KUKA KRL data list: CNC2.dat

&ACCESS RV
DEFDAT CNC2 Public
DECL GLOBAL FRAME gfCNCPoint2[30000]


gfCNCPoint2[1] = {X 204.1061, Y 40.0576, Z -2.1667, A 0.000, B 0.000, C 0.000 }
gfCNCPoint2[2] = {X 204.4089, Y 40.9162, Z -2.1667, A 0.000, B 0.000, C 0.000 }
gfCNCPoint2[3] = {X 204.5137, Y 41.8206, Z -2.1667, A 0.000, B 0.000, C 0.000 }
gfCNCPoint2[4] = {X 204.4154, Y 42.7257, Z -2.1667, A 0.000, B 0.000, C 0.000 }
gfCNCPoint2[5] = {X 204.1188, Y 43.5864, Z -2.1667, A 0.000, B 0.000, C 0.000 }
gfCNCPoint2[6] = {X 203.6387, Y 44.3600, Z -2.1667, A 0.000, B 0.000, C 0.000 }
gfCNCPoint2[7] = {X 202.9990, Y 45.0078, Z -2.1667, A 0.000, B 0.000, C 0.000 }
gfCNCPoint2[8] = {X 202.4628, Y 45.4414, Z -2.1667, A 0.000, B 0.000, C 0.000 }
gfCNCPoint2[9] = {X 201.7788, Y 45.8885, Z -2.1667, A 0.000, B 0.000, C 0.000 }
gfCNCPoint2[10] = {X 201.0196, Y 46.1910, Z -2.1667, A 0.000, B 0.000, C 0.000 }
gfCNCPoint2[11] = {X 200.2155, Y 46.3368, Z -2.1667, A 0.000, B 0.000, C 0.000 }
gfCNCPoint2[12] = {X 199.3985, Y 46.3200, Z -2.1667, A 0.000, B 0.000, C 0.000 }
gfCNCPoint2[13] = {X 198.6011, Y 46.1413, Z -2.1667, A 0.000, B 0.000, C 0.000 }
gfCNCPoint2[14] = {X 196.8579, Y 47.0738, Z -2.1667, A 0.000, B 0.000, C 0.000 }
gfCNCPoint2[15] = {X 195.0540, Y 47.8828, Z -2.1667, A 0.000, B 0.000, C 0.000 }
gfCNCPoint2[16] = {X 193.1983, Y 48.5643, Z -2.1667, A 0.000, B 0.000, C 0.000 }
gfCNCPoint2[17] = {X 191.2996, Y 49.1151, Z -2.1667, A 0.000, B 0.000, C 0.000 }
gfCNCPoint2[18] = {X 189.3771, Y 49.5045, Z -2.1667, A 0.000, B 0.000, C 0.000 }
gfCNCPoint2[19] = {X 187.4280, Y 49.7244, Z -2.1667, A 0.000, B 0.000, C 0.000 }
gfCNCPoint2[20] = {X 185.4671, Y 49.7730, Z -2.1667, A 0.000, B 0.000, C 0.000 }
gfCNCPoint2[21] = {X 183.5094, Y 49.6499, Z -2.1667, A 0.000, B 0.000, C 0.000 }
gfCNCPoint2[22] = {X 181.5700, Y 49.3561, Z -2.1667, A 0.000, B 0.000, C 0.000 }
gfCNCPoint2[23] = {X 179.7098, Y 48.8912, Z -2.1667, A 0.000, B 0.000, C 0.000 }
gfCNCPoint2[24] = {X 177.9148, Y 48.2172, Z -2.1667, A 0.000, B 0.000, C 0.000 }
gfCNCPoint2[25] = {X 176.2082, Y 47.3431, Z -2.1667, A 0.000, B 0.000, C 0.000 }
gfCNCPoint2[26] = {X 174.6124, Y 46.2802, Z -2.1667, A 0.000, B 0.000, C 0.000 }
gfCNCPoint2[27] = {X 173.4016, Y 45.2583, Z -2.1667, A 0.000, B 0.000, C 0.000 }
gfCNCPoint2[28] = {X 172.3241, Y 44.0965, Z -2.1667, A 0.000, B 0.000, C 0.000 }
gfCNCPoint2[29] = {X 171.3961, Y 42.8123, Z -2.1667, A 0.000, B 0.000, C 0.000 }
gfCNCPoint2[30] = {X 170.6313, Y 41.4246, Z -2.1667, A 0.000, B 0.000, C 0.000 }
gfCNCPoint2[31] = {X 170.0410, Y 39.9542, Z -2.1667, A 0.000, B 0.000, C 0.000 }
gfCNCPoint2[32] = {X 169.6341, Y 38.4229, Z -2.1667, A 0.000, B 0.000, C 0.000 }
gfCNCPoint2[33] = {X 169.4166, Y 36.8534, Z -2.1667, A 0.000, B 0.000, C 0.000 }
gfCNCPoint2[34] = {X 169.3333, Y 35.0485, Z -2.1667, A 0.000, B 0.000, C 0.000 }
gfCNCPoint2[35] = {X 169.4768, Y 33.2475, Z -2.1667, A 0.000, B 0.000, C 0.000 }
gfCNCPoint2[36] = {X 169.8448, Y 31.4786, Z -2.1667, A 0.000, B 0.000, C 0.000 }
gfCNCPoint2[37] = {X 170.4315, Y 29.7697, Z -2.1667, A 0.000, B 0.000, C 0.000 }
gfCNCPoint2[38] = {X 171.1150, Y 28.3909, Z -2.1667, A 0.000, B 0.000, C 0.000 }
gfCNCPoint2[39] = {X 171.9904, Y 27.1252, Z -2.1667, A 0.000, B 0.000, C 0.000 }
gfCNCPoint2[40] = {X 173.0396, Y 25.9993, Z -2.1667, A 0.000, B 0.000, C 0.000 }
gfCNCPoint2[41] = {X 174.2404, Y 25.0368, Z -2.1667, A 0.000, B 0.000, C 0.000 }
gfCNCPoint2[42] = {X 175.5677, Y 24.2579, Z -2.1667, A 0.000, B 0.000, C 0.000 }
gfCNCPoint2[43] = {X 174.6553, Y 23.9382, Z -2.1667, A 0.000, B 0.000, C 0.000 }
gfCNCPoint2[44] = {X 173.8439, Y 23.4129, Z -2.1667, A 0.000, B 0.000, C 0.000 }
gfCNCPoint2[45] = {X 173.1787, Y 22.7114, Z -2.1667, A 0.000, B 0.000, C 0.000 }
gfCNCPoint2[46] = {X 172.6973, Y 21.8731, Z -2.1667, A 0.000, B 0.000, C 0.000 }
gfCNCPoint2[47] = {X 171.3803, Y 18.6480, Z -2.1667, A 0.000, B 0.000, C 0.000 }
gfCNCPoint2[48] = {X 167.6770, Y 20.1603, Z -2.1667, A 0.000, B 0.000, C 0.000 }
gfCNCPoint2[49] = {X 167.6769, Y 20.1601, Z -2.1667, A 0.000, B 0.000, C 0.000 }
gfCNCPoint2[50] = {X 171.4542, Y 18.6179, Z -2.1667, A 0.000, B 0.000, C 0.000 }
gfCNCPoint2[51] = {X 170.1367, Y 15.3911, Z -2.1667, A 0.000, B 0.000, C 0.000 }
gfCNCPoint2[52] = {X 169.8835, Y 14.4675, Z -2.1667, A 0.000, B 0.000, C 0.000 }
gfCNCPoint2[53] = {X 169.8570, Y 13.5102, Z -2.1667, A 0.000, B 0.000, C 0.000 }
gfCNCPoint2[54] = {X 170.0588, Y 12.5740, Z -2.1667, A 0.000, B 0.000, C 0.000 }
gfCNCPoint2[55] = {X 170.4774, Y 11.7127, Z -2.1667, A 0.000, B 0.000, C 0.000 }
gfCNCPoint2[56] = {X 171.0888, Y 10.9755, Z -2.1667, A 0.000, B 0.000, C 0.000 }
gfCNCPoint2[57] = {X 171.8578, Y 10.4048, Z -2.1667, A 0.000, B 0.000, C 0.000 }
gfCNCPoint2[58] = {X 172.4867, Y 10.0462, Z -2.1667, A 0.000, B 0.000, C 0.000 }
gfCNCPoint2[59] = {X 173.3363, Y 9.6929, Z -2.1667, A 0.000, B 0.000, C 0.000 }
gfCNCPoint2[60] = {X 174.2443, Y 9.5431, Z -2.1667, A 0.000, B 0.000, C 0.000 }
gfCNCPoint2[61] = {X 175.1624, Y 9.6048, Z -2.1667, A 0.000, B 0.000, C 0.000 }
gfCNCPoint2[62] = {X 176.0421, Y 9.8746, Z -2.1667, A 0.000, B 0.000, C 0.000 }
gfCNCPoint2[63] = {X 178.2221, Y 8.9431, Z -2.1667, A 0.000, B 0.000, C 0.000 }
gfCNCPoint2[64] = {X 180.4850, Y 8.2365, Z -2.1667, A 0.000, B 0.000, C 0.000 }
gfCNCPoint2[65] = {X 182.8078, Y 7.7622, Z -2.1667, A 0.000, B 0.000, C 0.000 }
gfCNCPoint2[66] = {X 185.1665, Y 7.5249, Z -2.1667, A 0.000, B 0.000, C 0.000 }
gfCNCPoint2[67] = {X 187.5372, Y 7.5270, Z -2.1667, A 0.000, B 0.000, C 0.000 }
gfCNCPoint2[68] = {X 189.8955, Y 7.7686, Z -2.1667, A 0.000, B 0.000, C 0.000 }
gfCNCPoint2[69] = {X 191.6205, Y 8.1236, Z -2.1667, A 0.000, B 0.000, C 0.000 }
gfCNCPoint2[70] = {X 193.3000, Y 8.6537, Z -2.1667, A 0.000, B 0.000, C 0.000 }
gfCNCPoint2[71] = {X 194.9162, Y 9.3534, Z -2.1667, A 0.000, B 0.000, C 0.000 }
gfCNCPoint2[72] = {X 196.4521, Y 10.2153, Z -2.1667, A 0.000, B 0.000, C 0.000 }
gfCNCPoint2[73] = {X 197.8914, Y 11.2302, Z -2.1667, A 0.000, B 0.000, C 0.000 }
gfCNCPoint2[74] = {X 199.1662, Y 12.3971, Z -2.1667, A 0.000, B 0.000, C 0.000 }
gfCNCPoint2[75] = {X 200.2713, Y 13.7259, Z -2.1667, A 0.000, B 0.000, C 0.000 }
gfCNCPoint2[76] = {X 201.1862, Y 15.1921, Z -2.1667, A 0.000, B 0.000, C 0.000 }
gfCNCPoint2[77] = {X 201.8941, Y 16.7687, Z -2.1667, A 0.000, B 0.000, C 0.000 }
gfCNCPoint2[78] = {X 202.3577, Y 18.3894, Z -2.1667, A 0.000, B 0.000, C 0.000 }
gfCNCPoint2[79] = {X 202.6328, Y 20.0525, Z -2.1667, A 0.000, B 0.000, C 0.000 }
gfCNCPoint2[80] = {X 202.7157, Y 21.7361, Z -2.1667, A 0.000, B 0.000, C 0.000 }
gfCNCPoint2[81] = {X 202.6054, Y 23.4182, Z -2.1667, A 0.000, B 0.000, C 0.000 }
gfCNCPoint2[82] = {X 202.3032, Y 25.0766, Z -2.1667, A 0.000, B 0.000, C 0.000 }
gfCNCPoint2[83] = {X 201.8258, Y 26.6078, Z -2.1667, A 0.000, B 0.000, C 0.000 }
gfCNCPoint2[84] = {X 201.1376, Y 28.0565, Z -2.1667, A 0.000, B 0.000, C 0.000 }
gfCNCPoint2[85] = {X 200.2525, Y 29.3941, Z -2.1667, A 0.000, B 0.000, C 0.000 }
gfCNCPoint2[86] = {X 199.1879, Y 30.5938, Z -2.1667, A 0.000, B 0.000, C 0.000 }
gfCNCPoint2[87] = {X 197.9652, Y 31.6318, Z -2.1667, A 0.000, B 0.000, C 0.000 }
gfCNCPoint2[88] = {X 198.7272, Y 31.8156, Z -2.1667, A 0.000, B 0.000, C 0.000 }
gfCNCPoint2[89] = {X 199.4387, Y 32.1445, Z -2.1667, A 0.000, B 0.000, C 0.000 }
gfCNCPoint2[90] = {X 200.0724, Y 32.6059, Z -2.1667, A 0.000, B 0.000, C 0.000 }
gfCNCPoint2[91] = {X 200.6039, Y 33.1820, Z -2.1667, A 0.000, B 0.000, C 0.000 }
gfCNCPoint2[92] = {X 201.0129, Y 33.8507, Z -2.1667, A 0.000, B 0.000, C 0.000 }
gfCNCPoint2[93] = {X 204.0341, Y 40.0925, Z -2.1667, A 0.000, B 0.000, C 0.000 }
gfCNCPoint2[94] = {X 204.3309, Y 40.9342, Z -2.1667, A 0.000, B 0.000, C 0.000 }
gfCNCPoint2[95] = {X 204.4337, Y 41.8209, Z -2.1667, A 0.000, B 0.000, C 0.000 }
gfCNCPoint2[96] = {X 204.3373, Y 42.7082, Z -2.1667, A 0.000, B 0.000, C 0.000 }
gfCNCPoint2[97] = {X 204.0465, Y 43.5521, Z -2.1667, A 0.000, B 0.000, C 0.000 }
gfCNCPoint2[98] = {X 203.5758, Y 44.3105, Z -2.1667, A 0.000, B 0.000, C 0.000 }
gfCNCPoint2[99] = {X 202.9487, Y 44.9456, Z -2.1667, A 0.000, B 0.000, C 0.000 }
gfCNCPoint2[100] = {X 202.4125, Y 45.3791, Z -2.1667, A 0.000, B 0.000, C 0.000 }
gfCNCPoint2[101] = {X 201.7355, Y 45.8209, Z -2.1667, A 0.000, B 0.000, C 0.000 }
gfCNCPoint2[102] = {X 200.9837, Y 46.1181, Z -2.1667, A 0.000, B 0.000, C 0.000 }
gfCNCPoint2[103] = {X 200.1877, Y 46.2587, Z -2.1667, A 0.000, B 0.000, C 0.000 }
gfCNCPoint2[104] = {X 199.3796, Y 46.2370, Z -2.1667, A 0.000, B 0.000, C 0.000 }
gfCNCPoint2[105] = {X 198.5922, Y 46.0539, Z -2.1667, A 0.000, B 0.000, C 0.000 }
gfCNCPoint2[106] = {X 196.8470, Y 46.9900, Z -2.1667, A 0.000, B 0.000, C 0.000 }
gfCNCPoint2[107] = {X 195.0406, Y 47.8019, Z -2.1667, A 0.000, B 0.000, C 0.000 }
gfCNCPoint2[108] = {X 193.1819, Y 48.4855, Z -2.1667, A 0.000, B 0.000, C 0.000 }
gfCNCPoint2[109] = {X 191.2800, Y 49.0375, Z -2.1667, A 0.000, B 0.000, C 0.000 }
gfCNCPoint2[110] = {X 189.3644, Y 49.4255, Z -2.1667, A 0.000, B 0.000, C 0.000 }
gfCNCPoint2[111] = {X 187.4222, Y 49.6446, Z -2.1667, A 0.000, B 0.000, C 0.000 }
gfCNCPoint2[112] = {X 185.4683, Y 49.6930, Z -2.1667, A 0.000, B 0.000, C 0.000 }
gfCNCPoint2[113] = {X 183.5177, Y 49.5703, Z -2.1667, A 0.000, B 0.000, C 0.000 }
gfCNCPoint2[114] = {X 181.5852, Y 49.2775, Z -2.1667, A 0.000, B 0.000, C 0.000 }
gfCNCPoint2[115] = {X 179.7338, Y 48.8148, Z -2.1667, A 0.000, B 0.000, C 0.000 }
gfCNCPoint2[116] = {X 177.9472, Y 48.1441, Z -2.1667, A 0.000, B 0.000, C 0.000 }
gfCNCPoint2[117] = {X 176.2487, Y 47.2741, Z -2.1667, A 0.000, B 0.000, C 0.000 }
gfCNCPoint2[118] = {X 174.6604, Y 46.2162, Z -2.1667, A 0.000, B 0.000, C 0.000 }
gfCNCPoint2[119] = {X 173.4568, Y 45.2004, Z -2.1667, A 0.000, B 0.000, C 0.000 }
gfCNCPoint2[120] = {X 172.3859, Y 44.0456, Z -2.1667, A 0.000, B 0.000, C 0.000 }
gfCNCPoint2[121] = {X 171.4634, Y 42.7691, Z -2.1667, A 0.000, B 0.000, C 0.000 }
gfCNCPoint2[122] = {X 170.7033, Y 41.3898, Z -2.1667, A 0.000, B 0.000, C 0.000 }
gfCNCPoint2[123] = {X 170.1166, Y 39.9282, Z -2.1667, A 0.000, B 0.000, C 0.000 }
gfCNCPoint2[124] = {X 169.7123, Y 38.4060, Z -2.1667, A 0.000, B 0.000, C 0.000 }
gfCNCPoint2[125] = {X 169.4962, Y 36.8460, Z -2.1667, A 0.000, B 0.000, C 0.000 }
gfCNCPoint2[126] = {X 169.4132, Y 35.0508, Z -2.1667, A 0.000, B 0.000, C 0.000 }
gfCNCPoint2[127] = {X 169.5559, Y 33.2593, Z -2.1667, A 0.000, B 0.000, C 0.000 }
gfCNCPoint2[128] = {X 169.9219, Y 31.4998, Z -2.1667, A 0.000, B 0.000, C 0.000 }
gfCNCPoint2[129] = {X 170.5055, Y 29.8001, Z -2.1667, A 0.000, B 0.000, C 0.000 }
gfCNCPoint2[130] = {X 171.2085, Y 28.3899, Z -2.1667, A 0.000, B 0.000, C 0.000 }
gfCNCPoint2[131] = {X 172.1139, Y 27.1002, Z -2.1667, A 0.000, B 0.000, C 0.000 }
gfCNCPoint2[132] = {X 173.2013, Y 25.9598, Z -2.1667, A 0.000, B 0.000, C 0.000 }
gfCNCPoint2[133] = {X 174.4465, Y 24.9941, Z -2.1667, A 0.000, B 0.000, C 0.000 }
gfCNCPoint2[134] = {X 175.8218, Y 24.2249, Z -2.1667, A 0.000, B 0.000, C 0.000 }
gfCNCPoint2[135] = {X 175.0307, Y 24.0140, Z -2.1667, A 0.000, B 0.000, C 0.000 }
gfCNCPoint2[136] = {X 174.2991, Y 23.6464, Z -2.1667, A 0.000, B 0.000, C 0.000 }
gfCNCPoint2[137] = {X 173.6577, Y 23.1376, Z -2.1667, A 0.000, B 0.000, C 0.000 }
gfCNCPoint2[138] = {X 173.1333, Y 22.5089, Z -2.1667, A 0.000, B 0.000, C 0.000 }
gfCNCPoint2[139] = {X 172.7479, Y 21.7866, Z -2.1667, A 0.000, B 0.000, C 0.000 }
gfCNCPoint2[140] = {X 171.4542, Y 18.6179, Z -2.1667, A 0.000, B 0.000, C 0.000 }
gfCNCPoint2[141] = {X 167.6769, Y 20.1601, Z -2.1667, A 0.000, B 0.000, C 0.000 }
gfCNCPoint2[142] = {X 167.6769, Y 20.1601, Z 0.8333, A 0.000, B 0.000, C 0.000 }
gfCNCPoint2[143] = {X 167.6769, Y 20.1601, Z 11.0000, A 0.000, B 0.000, C 0.000 }
gfCNCPoint2[144] = {X 210.1659, Y 28.5742, Z 11.0000, A 0.000, B 0.000, C 0.000 }
gfCNCPoint2[145] = {X 210.1659, Y 28.5742, Z 0.8333, A 0.000, B 0.000, C 0.000 }
gfCNCPoint2[146] = {X 210.1659, Y 28.5742, Z -2.1667, A 0.000, B 0.000, C 0.000 }
gfCNCPoint2[147] = {X 214.2459, Y 28.5742, Z -2.1667, A 0.000, B 0.000, C 0.000 }
gfCNCPoint2[148] = {X 214.2459, Y 17.4624, Z -2.1667, A 0.000, B 0.000, C 0.000 }
gfCNCPoint2[149] = {X 214.2405, Y 16.7693, Z -2.1667, A 0.000, B 0.000, C 0.000 }
gfCNCPoint2[150] = {X 214.2433, Y 16.2731, Z -2.1667, A 0.000, B 0.000, C 0.000 }
gfCNCPoint2[151] = {X 213.6052, Y 15.6019, Z -2.1667, A 0.000, B 0.000, C 0.000 }
gfCNCPoint2[152] = {X 213.1248, Y 14.8101, Z -2.1667, A 0.000, B 0.000, C 0.000 }
gfCNCPoint2[153] = {X 212.8241, Y 13.9341, Z -2.1667, A 0.000, B 0.000, C 0.000 }
gfCNCPoint2[154] = {X 212.7172, Y 13.0141, Z -2.1667, A 0.000, B 0.000, C 0.000 }
gfCNCPoint2[155] = {X 212.7170, Y 12.1868, Z -2.1667, A 0.000, B 0.000, C 0.000 }
gfCNCPoint2[156] = {X 212.8253, Y 11.2255, Z -2.1667, A 0.000, B 0.000, C 0.000 }
gfCNCPoint2[157] = {X 213.1448, Y 10.3124, Z -2.1667, A 0.000, B 0.000, C 0.000 }
gfCNCPoint2[158] = {X 213.6595, Y 9.4933, Z -2.1667, A 0.000, B 0.000, C 0.000 }
gfCNCPoint2[159] = {X 214.3435, Y 8.8093, Z -2.1667, A 0.000, B 0.000, C 0.000 }
gfCNCPoint2[160] = {X 215.1626, Y 8.2946, Z -2.1667, A 0.000, B 0.000, C 0.000 }
gfCNCPoint2[161] = {X 216.0757, Y 7.9751, Z -2.1667, A 0.000, B 0.000, C 0.000 }
gfCNCPoint2[162] = {X 217.0370, Y 7.8668, Z -2.1667, A 0.000, B 0.000, C 0.000 }
gfCNCPoint2[163] = {X 223.4805, Y 7.8668, Z -2.1667, A 0.000, B 0.000, C 0.000 }
gfCNCPoint2[164] = {X 224.4418, Y 7.9751, Z -2.1667, A 0.000, B 0.000, C 0.000 }
gfCNCPoint2[165] = {X 225.3549, Y 8.2946, Z -2.1667, A 0.000, B 0.000, C 0.000 }
gfCNCPoint2[166] = {X 226.1740, Y 8.8093, Z -2.1667, A 0.000, B 0.000, C 0.000 }
gfCNCPoint2[167] = {X 226.8580, Y 9.4933, Z -2.1667, A 0.000, B 0.000, C 0.000 }
gfCNCPoint2[168] = {X 227.3727, Y 10.3124, Z -2.1667, A 0.000, B 0.000, C 0.000 }
gfCNCPoint2[169] = {X 227.6922, Y 11.2255, Z -2.1667, A 0.000, B 0.000, C 0.000 }
gfCNCPoint2[170] = {X 227.8005, Y 12.1868, Z -2.1667, A 0.000, B 0.000, C 0.000 }
gfCNCPoint2[171] = {X 227.8005, Y 12.9781, Z -2.1667, A 0.000, B 0.000, C 0.000 }
gfCNCPoint2[172] = {X 227.6991, Y 13.9083, Z -2.1667, A 0.000, B 0.000, C 0.000 }
gfCNCPoint2[173] = {X 227.3998, Y 14.7949, Z -2.1667, A 0.000, B 0.000, C 0.000 }
gfCNCPoint2[174] = {X 226.9167, Y 15.5962, Z -2.1667, A 0.000, B 0.000, C 0.000 }
gfCNCPoint2[175] = {X 226.2723, Y 16.2747, Z -2.1667, A 0.000, B 0.000, C 0.000 }
gfCNCPoint2[176] = {X 226.2732, Y 40.9153, Z -2.1667, A 0.000, B 0.000, C 0.000 }
gfCNCPoint2[177] = {X 226.9108, Y 41.5854, Z -2.1667, A 0.000, B 0.000, C 0.000 }
gfCNCPoint2[178] = {X 227.3912, Y 42.3758, Z -2.1667, A 0.000, B 0.000, C 0.000 }
gfCNCPoint2[179] = {X 227.6923, Y 43.2503, Z -2.1667, A 0.000, B 0.000, C 0.000 }
gfCNCPoint2[180] = {X 227.8003, Y 44.1689, Z -2.1667, A 0.000, B 0.000, C 0.000 }
gfCNCPoint2[181] = {X 227.8005, Y 45.0000, Z -2.1667, A 0.000, B 0.000, C 0.000 }
gfCNCPoint2[182] = {X 227.6922, Y 45.9613, Z -2.1667, A 0.000, B 0.000, C 0.000 }
gfCNCPoint2[183] = {X 227.3727, Y 46.8744, Z -2.1667, A 0.000, B 0.000, C 0.000 }
gfCNCPoint2[184] = {X 226.8580, Y 47.6935, Z -2.1667, A 0.000, B 0.000, C 0.000 }
gfCNCPoint2[185] = {X 226.1740, Y 48.3775, Z -2.1667, A 0.000, B 0.000, C 0.000 }
gfCNCPoint2[186] = {X 225.3549, Y 48.8922, Z -2.1667, A 0.000, B 0.000, C 0.000 }
gfCNCPoint2[187] = {X 224.4418, Y 49.2117, Z -2.1667, A 0.000, B 0.000, C 0.000 }
gfCNCPoint2[188] = {X 223.4805, Y 49.3200, Z -2.1667, A 0.000, B 0.000, C 0.000 }
gfCNCPoint2[189] = {X 217.0370, Y 49.3200, Z -2.1667, A 0.000, B 0.000, C 0.000 }
gfCNCPoint2[190] = {X 216.0805, Y 49.2128, Z -2.1667, A 0.000, B 0.000, C 0.000 }
gfCNCPoint2[191] = {X 215.1715, Y 48.8964, Z -2.1667, A 0.000, B 0.000, C 0.000 }
gfCNCPoint2[192] = {X 214.3551, Y 48.3867, Z -2.1667, A 0.000, B 0.000, C 0.000 }
gfCNCPoint2[193] = {X 213.6718, Y 47.7088, Z -2.1667, A 0.000, B 0.000, C 0.000 }
gfCNCPoint2[194] = {X 213.1556, Y 46.8965, Z -2.1667, A 0.000, B 0.000, C 0.000 }
gfCNCPoint2[195] = {X 212.8320, Y 45.9901, Z -2.1667, A 0.000, B 0.000, C 0.000 }
gfCNCPoint2[196] = {X 212.7172, Y 45.0345, Z -2.1667, A 0.000, B 0.000, C 0.000 }
gfCNCPoint2[197] = {X 212.7170, Y 44.1994, Z -2.1667, A 0.000, B 0.000, C 0.000 }
gfCNCPoint2[198] = {X 212.7890, Y 43.4200, Z -2.1667, A 0.000, B 0.000, C 0.000 }
gfCNCPoint2[199] = {X 213.0024, Y 42.6670, Z -2.1667, A 0.000, B 0.000, C 0.000 }
gfCNCPoint2[200] = {X 213.3500, Y 41.9658, Z -2.1667, A 0.000, B 0.000, C 0.000 }
gfCNCPoint2[201] = {X 213.8202, Y 41.3400, Z -2.1667, A 0.000, B 0.000, C 0.000 }
gfCNCPoint2[202] = {X 214.2415, Y 40.8754, Z -2.1667, A 0.000, B 0.000, C 0.000 }
gfCNCPoint2[203] = {X 214.2459, Y 40.3062, Z -2.1667, A 0.000, B 0.000, C 0.000 }
gfCNCPoint2[204] = {X 214.2459, Y 28.5742, Z -2.1667, A 0.000, B 0.000, C 0.000 }
gfCNCPoint2[205] = {X 210.2459, Y 28.5742, Z -2.1667, A 0.000, B 0.000, C 0.000 }
gfCNCPoint2[206] = {X 214.3259, Y 28.5742, Z -2.1667, A 0.000, B 0.000, C 0.000 }
gfCNCPoint2[207] = {X 214.3259, Y 17.4621, Z -2.1667, A 0.000, B 0.000, C 0.000 }
gfCNCPoint2[208] = {X 214.3205, Y 16.7693, Z -2.1667, A 0.000, B 0.000, C 0.000 }
gfCNCPoint2[209] = {X 214.3235, Y 16.2360, Z -2.1667, A 0.000, B 0.000, C 0.000 }
gfCNCPoint2[210] = {X 213.6857, Y 15.5754, Z -2.1667, A 0.000, B 0.000, C 0.000 }
gfCNCPoint2[211] = {X 213.2051, Y 14.7930, Z -2.1667, A 0.000, B 0.000, C 0.000 }
gfCNCPoint2[212] = {X 212.9042, Y 13.9255, Z -2.1667, A 0.000, B 0.000, C 0.000 }
gfCNCPoint2[213] = {X 212.7972, Y 13.0135, Z -2.1667, A 0.000, B 0.000, C 0.000 }
gfCNCPoint2[214] = {X 212.7970, Y 12.1868, Z -2.1667, A 0.000, B 0.000, C 0.000 }
gfCNCPoint2[215] = {X 212.9033, Y 11.2433, Z -2.1667, A 0.000, B 0.000, C 0.000 }
gfCNCPoint2[216] = {X 213.2169, Y 10.3472, Z -2.1667, A 0.000, B 0.000, C 0.000 }
gfCNCPoint2[217] = {X 213.7220, Y 9.5432, Z -2.1667, A 0.000, B 0.000, C 0.000 }
gfCNCPoint2[218] = {X 214.3934, Y 8.8719, Z -2.1667, A 0.000, B 0.000, C 0.000 }
gfCNCPoint2[219] = {X 215.1973, Y 8.3667, Z -2.1667, A 0.000, B 0.000, C 0.000 }
gfCNCPoint2[220] = {X 216.0935, Y 8.0531, Z -2.1667, A 0.000, B 0.000, C 0.000 }
gfCNCPoint2[221] = {X 217.0370, Y 7.9468, Z -2.1667, A 0.000, B 0.000, C 0.000 }
gfCNCPoint2[222] = {X 223.4805, Y 7.9468, Z -2.1667, A 0.000, B 0.000, C 0.000 }
gfCNCPoint2[223] = {X 224.4240, Y 8.0531, Z -2.1667, A 0.000, B 0.000, C 0.000 }
gfCNCPoint2[224] = {X 225.3201, Y 8.3667, Z -2.1667, A 0.000, B 0.000, C 0.000 }
gfCNCPoint2[225] = {X 226.1241, Y 8.8718, Z -2.1667, A 0.000, B 0.000, C 0.000 }
gfCNCPoint2[226] = {X 226.7954, Y 9.5432, Z -2.1667, A 0.000, B 0.000, C 0.000 }
gfCNCPoint2[227] = {X 227.3006, Y 10.3471, Z -2.1667, A 0.000, B 0.000, C 0.000 }
gfCNCPoint2[228] = {X 227.6142, Y 11.2433, Z -2.1667, A 0.000, B 0.000, C 0.000 }
gfCNCPoint2[229] = {X 227.7205, Y 12.1868, Z -2.1667, A 0.000, B 0.000, C 0.000 }
gfCNCPoint2[230] = {X 227.7205, Y 12.9781, Z -2.1667, A 0.000, B 0.000, C 0.000 }
gfCNCPoint2[231] = {X 227.6190, Y 13.9001, Z -2.1667, A 0.000, B 0.000, C 0.000 }
gfCNCPoint2[232] = {X 227.3195, Y 14.7780, Z -2.1667, A 0.000, B 0.000, C 0.000 }
gfCNCPoint2[233] = {X 226.8362, Y 15.5697, Z -2.1667, A 0.000, B 0.000, C 0.000 }
gfCNCPoint2[234] = {X 226.1923, Y 16.2374, Z -2.1667, A 0.000, B 0.000, C 0.000 }
gfCNCPoint2[235] = {X 226.1932, Y 40.9526, Z -2.1667, A 0.000, B 0.000, C 0.000 }
gfCNCPoint2[236] = {X 226.8304, Y 41.6121, Z -2.1667, A 0.000, B 0.000, C 0.000 }
gfCNCPoint2[237] = {X 227.3109, Y 42.3931, Z -2.1667, A 0.000, B 0.000, C 0.000 }
gfCNCPoint2[238] = {X 227.6122, Y 43.2591, Z -2.1667, A 0.000, B 0.000, C 0.000 }
gfCNCPoint2[239] = {X 227.7203, Y 44.1697, Z -2.1667, A 0.000, B 0.000, C 0.000 }
gfCNCPoint2[240] = {X 227.7205, Y 45.0000, Z -2.1667, A 0.000, B 0.000, C 0.000 }
gfCNCPoint2[241] = {X 227.6142, Y 45.9435, Z -2.1667, A 0.000, B 0.000, C 0.000 }
gfCNCPoint2[242] = {X 227.3006, Y 46.8397, Z -2.1667, A 0.000, B 0.000, C 0.000 }
gfCNCPoint2[243] = {X 226.7954, Y 47.6436, Z -2.1667, A 0.000, B 0.000, C 0.000 }
gfCNCPoint2[244] = {X 226.1241, Y 48.3150, Z -2.1667, A 0.000, B 0.000, C 0.000 }
gfCNCPoint2[245] = {X 225.3201, Y 48.8201, Z -2.1667, A 0.000, B 0.000, C 0.000 }
gfCNCPoint2[246] = {X 224.4240, Y 49.1337, Z -2.1667, A 0.000, B 0.000, C 0.000 }
gfCNCPoint2[247] = {X 223.4805, Y 49.2400, Z -2.1667, A 0.000, B 0.000, C 0.000 }
gfCNCPoint2[248] = {X 217.0370, Y 49.2400, Z -2.1667, A 0.000, B 0.000, C 0.000 }
gfCNCPoint2[249] = {X 216.0982, Y 49.1348, Z -2.1667, A 0.000, B 0.000, C 0.000 }
gfCNCPoint2[250] = {X 215.2061, Y 48.8243, Z -2.1667, A 0.000, B 0.000, C 0.000 }
gfCNCPoint2[251] = {X 214.4048, Y 48.3240, Z -2.1667, A 0.000, B 0.000, C 0.000 }
gfCNCPoint2[252] = {X 213.7341, Y 47.6587, Z -2.1667, A 0.000, B 0.000, C 0.000 }
gfCNCPoint2[253] = {X 213.2275, Y 46.8614, Z -2.1667, A 0.000, B 0.000, C 0.000 }
gfCNCPoint2[254] = {X 212.9099, Y 45.9717, Z -2.1667, A 0.000, B 0.000, C 0.000 }
gfCNCPoint2[255] = {X 212.7972, Y 45.0338, Z -2.1667, A 0.000, B 0.000, C 0.000 }
gfCNCPoint2[256] = {X 212.7970, Y 44.1994, Z -2.1667, A 0.000, B 0.000, C 0.000 }
gfCNCPoint2[257] = {X 212.8676, Y 43.4347, Z -2.1667, A 0.000, B 0.000, C 0.000 }
gfCNCPoint2[258] = {X 213.0770, Y 42.6958, Z -2.1667, A 0.000, B 0.000, C 0.000 }
gfCNCPoint2[259] = {X 213.4181, Y 42.0077, Z -2.1667, A 0.000, B 0.000, C 0.000 }
gfCNCPoint2[260] = {X 213.8795, Y 41.3938, Z -2.1667, A 0.000, B 0.000, C 0.000 }
gfCNCPoint2[261] = {X 214.3213, Y 40.9065, Z -2.1667, A 0.000, B 0.000, C 0.000 }
gfCNCPoint2[262] = {X 214.3259, Y 40.3065, Z -2.1667, A 0.000, B 0.000, C 0.000 }
gfCNCPoint2[263] = {X 214.3259, Y 28.5742, Z -2.1667, A 0.000, B 0.000, C 0.000 }
gfCNCPoint2[264] = {X 210.3259, Y 28.5742, Z -2.1667, A 0.000, B 0.000, C 0.000 }
gfCNCPoint2[265] = {X 214.4059, Y 28.5742, Z -2.1667, A 0.000, B 0.000, C 0.000 }
gfCNCPoint2[266] = {X 214.4059, Y 17.4618, Z -2.1667, A 0.000, B 0.000, C 0.000 }
gfCNCPoint2[267] = {X 214.4005, Y 16.7692, Z -2.1667, A 0.000, B 0.000, C 0.000 }
gfCNCPoint2[268] = {X 214.4038, Y 16.1985, Z -2.1667, A 0.000, B 0.000, C 0.000 }
gfCNCPoint2[269] = {X 213.7663, Y 15.5487, Z -2.1667, A 0.000, B 0.000, C 0.000 }
gfCNCPoint2[270] = {X 213.2855, Y 14.7758, Z -2.1667, A 0.000, B 0.000, C 0.000 }
gfCNCPoint2[271] = {X 212.9843, Y 13.9168, Z -2.1667, A 0.000, B 0.000, C 0.000 }
gfCNCPoint2[272] = {X 212.8772, Y 13.0128, Z -2.1667, A 0.000, B 0.000, C 0.000 }
gfCNCPoint2[273] = {X 212.8770, Y 12.1868, Z -2.1667, A 0.000, B 0.000, C 0.000 }
gfCNCPoint2[274] = {X 212.9813, Y 11.2611, Z -2.1667, A 0.000, B 0.000, C 0.000 }
gfCNCPoint2[275] = {X 213.2890, Y 10.3819, Z -2.1667, A 0.000, B 0.000, C 0.000 }
gfCNCPoint2[276] = {X 213.7846, Y 9.5931, Z -2.1667, A 0.000, B 0.000, C 0.000 }
gfCNCPoint2[277] = {X 214.4433, Y 8.9344, Z -2.1667, A 0.000, B 0.000, C 0.000 }
gfCNCPoint2[278] = {X 215.2321, Y 8.4388, Z -2.1667, A 0.000, B 0.000, C 0.000 }
gfCNCPoint2[279] = {X 216.1113, Y 8.1311, Z -2.1667, A 0.000, B 0.000, C 0.000 }
gfCNCPoint2[280] = {X 217.0370, Y 8.0268, Z -2.1667, A 0.000, B 0.000, C 0.000 }
gfCNCPoint2[281] = {X 223.4805, Y 8.0268, Z -2.1667, A 0.000, B 0.000, C 0.000 }
gfCNCPoint2[282] = {X 224.4062, Y 8.1311, Z -2.1667, A 0.000, B 0.000, C 0.000 }
gfCNCPoint2[283] = {X 225.2854, Y 8.4388, Z -2.1667, A 0.000, B 0.000, C 0.000 }
gfCNCPoint2[284] = {X 226.0742, Y 8.9344, Z -2.1667, A 0.000, B 0.000, C 0.000 }
gfCNCPoint2[285] = {X 226.7329, Y 9.5931, Z -2.1667, A 0.000, B 0.000, C 0.000 }
gfCNCPoint2[286] = {X 227.2285, Y 10.3819, Z -2.1667, A 0.000, B 0.000, C 0.000 }
gfCNCPoint2[287] = {X 227.5362, Y 11.2611, Z -2.1667, A 0.000, B 0.000, C 0.000 }
gfCNCPoint2[288] = {X 227.6405, Y 12.1868, Z -2.1667, A 0.000, B 0.000, C 0.000 }
gfCNCPoint2[289] = {X 227.6405, Y 12.9781, Z -2.1667, A 0.000, B 0.000, C 0.000 }
gfCNCPoint2[290] = {X 227.5389, Y 13.8918, Z -2.1667, A 0.000, B 0.000, C 0.000 }
gfCNCPoint2[291] = {X 227.2391, Y 14.7609, Z -2.1667, A 0.000, B 0.000, C 0.000 }
gfCNCPoint2[292] = {X 226.7557, Y 15.5429, Z -2.1667, A 0.000, B 0.000, C 0.000 }
gfCNCPoint2[293] = {X 226.1123, Y 16.1997, Z -2.1667, A 0.000, B 0.000, C 0.000 }
gfCNCPoint2[294] = {X 226.1132, Y 40.9903, Z -2.1667, A 0.000, B 0.000, C 0.000 }
gfCNCPoint2[295] = {X 226.7499, Y 41.6390, Z -2.1667, A 0.000, B 0.000, C 0.000 }
gfCNCPoint2[296] = {X 227.2306, Y 42.4105, Z -2.1667, A 0.000, B 0.000, C 0.000 }
gfCNCPoint2[297] = {X 227.5321, Y 43.2680, Z -2.1667, A 0.000, B 0.000, C 0.000 }
gfCNCPoint2[298] = {X 227.6403, Y 44.1704, Z -2.1667, A 0.000, B 0.000, C 0.000 }
gfCNCPoint2[299] = {X 227.6405, Y 45.0000, Z -2.1667, A 0.000, B 0.000, C 0.000 }
gfCNCPoint2[300] = {X 227.5362, Y 45.9257, Z -2.1667, A 0.000, B 0.000, C 0.000 }
gfCNCPoint2[301] = {X 227.2285, Y 46.8050, Z -2.1667, A 0.000, B 0.000, C 0.000 }
gfCNCPoint2[302] = {X 226.7329, Y 47.5937, Z -2.1667, A 0.000, B 0.000, C 0.000 }
gfCNCPoint2[303] = {X 226.0742, Y 48.2524, Z -2.1667, A 0.000, B 0.000, C 0.000 }
gfCNCPoint2[304] = {X 225.2854, Y 48.7480, Z -2.1667, A 0.000, B 0.000, C 0.000 }
gfCNCPoint2[305] = {X 224.4062, Y 49.0557, Z -2.1667, A 0.000, B 0.000, C 0.000 }
gfCNCPoint2[306] = {X 223.4805, Y 49.1600, Z -2.1667, A 0.000, B 0.000, C 0.000 }
gfCNCPoint2[307] = {X 217.0370, Y 49.1600, Z -2.1667, A 0.000, B 0.000, C 0.000 }
gfCNCPoint2[308] = {X 216.1160, Y 49.0568, Z -2.1667, A 0.000, B 0.000, C 0.000 }
gfCNCPoint2[309] = {X 215.2406, Y 48.7521, Z -2.1667, A 0.000, B 0.000, C 0.000 }
gfCNCPoint2[310] = {X 214.4544, Y 48.2613, Z -2.1667, A 0.000, B 0.000, C 0.000 }
gfCNCPoint2[311] = {X 213.7965, Y 47.6085, Z -2.1667, A 0.000, B 0.000, C 0.000 }
gfCNCPoint2[312] = {X 213.2993, Y 46.8263, Z -2.1667, A 0.000, B 0.000, C 0.000 }
gfCNCPoint2[313] = {X 212.9877, Y 45.9534, Z -2.1667, A 0.000, B 0.000, C 0.000 }
gfCNCPoint2[314] = {X 212.8771, Y 45.0332, Z -2.1667, A 0.000, B 0.000, C 0.000 }
gfCNCPoint2[315] = {X 212.8770, Y 44.1994, Z -2.1667, A 0.000, B 0.000, C 0.000 }
gfCNCPoint2[316] = {X 212.9463, Y 43.4493, Z -2.1667, A 0.000, B 0.000, C 0.000 }
gfCNCPoint2[317] = {X 213.1517, Y 42.7246, Z -2.1667, A 0.000, B 0.000, C 0.000 }
gfCNCPoint2[318] = {X 213.4863, Y 42.0497, Z -2.1667, A 0.000, B 0.000, C 0.000 }
gfCNCPoint2[319] = {X 213.9387, Y 41.4475, Z -2.1667, A 0.000, B 0.000, C 0.000 }
gfCNCPoint2[320] = {X 214.4010, Y 40.9376, Z -2.1667, A 0.000, B 0.000, C 0.000 }
gfCNCPoint2[321] = {X 214.4059, Y 40.3068, Z -2.1667, A 0.000, B 0.000, C 0.000 }
gfCNCPoint2[322] = {X 214.4059, Y 28.5742, Z -2.1667, A 0.000, B 0.000, C 0.000 }
gfCNCPoint2[323] = {X 210.4059, Y 28.5742, Z -2.1667, A 0.000, B 0.000, C 0.000 }
gfCNCPoint2[324] = {X 214.4859, Y 28.5742, Z -2.1667, A 0.000, B 0.000, C 0.000 }
gfCNCPoint2[325] = {X 214.4859, Y 17.4614, Z -2.1667, A 0.000, B 0.000, C 0.000 }
gfCNCPoint2[326] = {X 214.4805, Y 16.7691, Z -2.1667, A 0.000, B 0.000, C 0.000 }
gfCNCPoint2[327] = {X 214.4840, Y 16.1605, Z -2.1667, A 0.000, B 0.000, C 0.000 }
gfCNCPoint2[328] = {X 214.4262, Y 16.1133, Z -2.1667, A 0.000, B 0.000, C 0.000 }
gfCNCPoint2[329] = {X 214.3692, Y 16.0650, Z -2.1667, A 0.000, B 0.000, C 0.000 }
gfCNCPoint2[330] = {X 213.7783, Y 15.4331, Z -2.1667, A 0.000, B 0.000, C 0.000 }
gfCNCPoint2[331] = {X 213.3340, Y 14.6908, Z -2.1667, A 0.000, B 0.000, C 0.000 }
gfCNCPoint2[332] = {X 213.0561, Y 13.8716, Z -2.1667, A 0.000, B 0.000, C 0.000 }
gfCNCPoint2[333] = {X 212.9572, Y 13.0121, Z -2.1667, A 0.000, B 0.000, C 0.000 }
gfCNCPoint2[334] = {X 212.9570, Y 12.1868, Z -2.1667, A 0.000, B 0.000, C 0.000 }
gfCNCPoint2[335] = {X 213.0593, Y 11.2789, Z -2.1667, A 0.000, B 0.000, C 0.000 }
gfCNCPoint2[336] = {X 213.3611, Y 10.4166, Z -2.1667, A 0.000, B 0.000, C 0.000 }
gfCNCPoint2[337] = {X 213.8471, Y 9.6430, Z -2.1667, A 0.000, B 0.000, C 0.000 }
gfCNCPoint2[338] = {X 214.4932, Y 8.9969, Z -2.1667, A 0.000, B 0.000, C 0.000 }
gfCNCPoint2[339] = {X 215.2668, Y 8.5109, Z -2.1667, A 0.000, B 0.000, C 0.000 }
gfCNCPoint2[340] = {X 216.1291, Y 8.2091, Z -2.1667, A 0.000, B 0.000, C 0.000 }
gfCNCPoint2[341] = {X 217.0370, Y 8.1068, Z -2.1667, A 0.000, B 0.000, C 0.000 }
gfCNCPoint2[342] = {X 223.4805, Y 8.1068, Z -2.1667, A 0.000, B 0.000, C 0.000 }
gfCNCPoint2[343] = {X 224.3884, Y 8.2091, Z -2.1667, A 0.000, B 0.000, C 0.000 }
gfCNCPoint2[344] = {X 225.2507, Y 8.5109, Z -2.1667, A 0.000, B 0.000, C 0.000 }
gfCNCPoint2[345] = {X 226.0243, Y 8.9969, Z -2.1667, A 0.000, B 0.000, C 0.000 }
gfCNCPoint2[346] = {X 226.6704, Y 9.6430, Z -2.1667, A 0.000, B 0.000, C 0.000 }
gfCNCPoint2[347] = {X 227.1564, Y 10.4166, Z -2.1667, A 0.000, B 0.000, C 0.000 }
gfCNCPoint2[348] = {X 227.4582, Y 11.2789, Z -2.1667, A 0.000, B 0.000, C 0.000 }
gfCNCPoint2[349] = {X 227.5605, Y 12.1868, Z -2.1667, A 0.000, B 0.000, C 0.000 }
gfCNCPoint2[350] = {X 227.5605, Y 12.9781, Z -2.1667, A 0.000, B 0.000, C 0.000 }
gfCNCPoint2[351] = {X 227.4587, Y 13.8835, Z -2.1667, A 0.000, B 0.000, C 0.000 }
gfCNCPoint2[352] = {X 227.1586, Y 14.7437, Z -2.1667, A 0.000, B 0.000, C 0.000 }
gfCNCPoint2[353] = {X 226.6751, Y 15.5159, Z -2.1667, A 0.000, B 0.000, C 0.000 }
gfCNCPoint2[354] = {X 226.0323, Y 16.1615, Z -2.1667, A 0.000, B 0.000, C 0.000 }
gfCNCPoint2[355] = {X 226.0332, Y 41.0286, Z -2.1667, A 0.000, B 0.000, C 0.000 }
gfCNCPoint2[356] = {X 226.1409, Y 41.1154, Z -2.1667, A 0.000, B 0.000, C 0.000 }
gfCNCPoint2[357] = {X 226.7342, Y 41.7472, Z -2.1667, A 0.000, B 0.000, C 0.000 }
gfCNCPoint2[358] = {X 227.1807, Y 42.4899, Z -2.1667, A 0.000, B 0.000, C 0.000 }
gfCNCPoint2[359] = {X 227.4603, Y 43.3103, Z -2.1667, A 0.000, B 0.000, C 0.000 }
gfCNCPoint2[360] = {X 227.5603, Y 44.1712, Z -2.1667, A 0.000, B 0.000, C 0.000 }
gfCNCPoint2[361] = {X 227.5605, Y 45.0000, Z -2.1667, A 0.000, B 0.000, C 0.000 }
gfCNCPoint2[362] = {X 227.4582, Y 45.9079, Z -2.1667, A 0.000, B 0.000, C 0.000 }
gfCNCPoint2[363] = {X 227.1564, Y 46.7702, Z -2.1667, A 0.000, B 0.000, C 0.000 }
gfCNCPoint2[364] = {X 226.6704, Y 47.5438, Z -2.1667, A 0.000, B 0.000, C 0.000 }
gfCNCPoint2[365] = {X 226.0243, Y 48.1899, Z -2.1667, A 0.000, B 0.000, C 0.000 }
gfCNCPoint2[366] = {X 225.2507, Y 48.6760, Z -2.1667, A 0.000, B 0.000, C 0.000 }
gfCNCPoint2[367] = {X 224.3884, Y 48.9777, Z -2.1667, A 0.000, B 0.000, C 0.000 }
gfCNCPoint2[368] = {X 223.4805, Y 49.0800, Z -2.1667, A 0.000, B 0.000, C 0.000 }
gfCNCPoint2[369] = {X 217.0370, Y 49.0800, Z -2.1667, A 0.000, B 0.000, C 0.000 }
gfCNCPoint2[370] = {X 216.1337, Y 48.9787, Z -2.1667, A 0.000, B 0.000, C 0.000 }
gfCNCPoint2[371] = {X 215.2752, Y 48.6800, Z -2.1667, A 0.000, B 0.000, C 0.000 }
gfCNCPoint2[372] = {X 214.5041, Y 48.1986, Z -2.1667, A 0.000, B 0.000, C 0.000 }
gfCNCPoint2[373] = {X 213.8588, Y 47.5584, Z -2.1667, A 0.000, B 0.000, C 0.000 }
gfCNCPoint2[374] = {X 213.3712, Y 46.7912, Z -2.1667, A 0.000, B 0.000, C 0.000 }
gfCNCPoint2[375] = {X 213.0656, Y 45.9351, Z -2.1667, A 0.000, B 0.000, C 0.000 }
gfCNCPoint2[376] = {X 212.9571, Y 45.0325, Z -2.1667, A 0.000, B 0.000, C 0.000 }
gfCNCPoint2[377] = {X 212.9570, Y 44.1994, Z -2.1667, A 0.000, B 0.000, C 0.000 }
gfCNCPoint2[378] = {X 213.0249, Y 43.4640, Z -2.1667, A 0.000, B 0.000, C 0.000 }
gfCNCPoint2[379] = {X 213.2263, Y 42.7534, Z -2.1667, A 0.000, B 0.000, C 0.000 }
gfCNCPoint2[380] = {X 213.5544, Y 42.0917, Z -2.1667, A 0.000, B 0.000, C 0.000 }
gfCNCPoint2[381] = {X 213.9980, Y 41.5012, Z -2.1667, A 0.000, B 0.000, C 0.000 }
gfCNCPoint2[382] = {X 214.4808, Y 40.9687, Z -2.1667, A 0.000, B 0.000, C 0.000 }
gfCNCPoint2[383] = {X 214.4859, Y 40.3072, Z -2.1667, A 0.000, B 0.000, C 0.000 }
gfCNCPoint2[384] = {X 214.4859, Y 28.5742, Z -2.1667, A 0.000, B 0.000, C 0.000 }
gfCNCPoint2[385] = {X 210.4859, Y 28.5742, Z -2.1667, A 0.000, B 0.000, C 0.000 }
gfCNCPoint2[386] = {X 214.5659, Y 28.5742, Z -2.1667, A 0.000, B 0.000, C 0.000 }
gfCNCPoint2[387] = {X 214.5659, Y 17.4611, Z -2.1667, A 0.000, B 0.000, C 0.000 }
gfCNCPoint2[388] = {X 214.5605, Y 16.7687, Z -2.1667, A 0.000, B 0.000, C 0.000 }
gfCNCPoint2[389] = {X 214.5598, Y 16.1862, Z -2.1667, A 0.000, B 0.000, C 0.000 }
gfCNCPoint2[390] = {X 214.5756, Y 16.1310, Z -2.1667, A 0.000, B 0.000, C 0.000 }
gfCNCPoint2[391] = {X 214.4978, Y 16.0687, Z -2.1667, A 0.000, B 0.000, C 0.000 }
gfCNCPoint2[392] = {X 214.4215, Y 16.0044, Z -2.1667, A 0.000, B 0.000, C 0.000 }
gfCNCPoint2[393] = {X 213.8372, Y 15.3783, Z -2.1667, A 0.000, B 0.000, C 0.000 }
gfCNCPoint2[394] = {X 213.3996, Y 14.6420, Z -2.1667, A 0.000, B 0.000, C 0.000 }
gfCNCPoint2[395] = {X 213.1287, Y 13.8295, Z -2.1667, A 0.000, B 0.000, C 0.000 }
gfCNCPoint2[396] = {X 213.0370, Y 12.9779, Z -2.1667, A 0.000, B 0.000, C 0.000 }
gfCNCPoint2[397] = {X 213.0370, Y 12.1868, Z -2.1667, A 0.000, B 0.000, C 0.000 }
gfCNCPoint2[398] = {X 213.1373, Y 11.2967, Z -2.1667, A 0.000, B 0.000, C 0.000 }
gfCNCPoint2[399] = {X 213.4331, Y 10.4513, Z -2.1667, A 0.000, B 0.000, C 0.000 }
gfCNCPoint2[400] = {X 213.9097, Y 9.6929, Z -2.1667, A 0.000, B 0.000, C 0.000 }
gfCNCPoint2[401] = {X 214.5431, Y 9.0595, Z -2.1667, A 0.000, B 0.000, C 0.000 }
gfCNCPoint2[402] = {X 215.3015, Y 8.5829, Z -2.1667, A 0.000, B 0.000, C 0.000 }
gfCNCPoint2[403] = {X 216.1469, Y 8.2871, Z -2.1667, A 0.000, B 0.000, C 0.000 }
gfCNCPoint2[404] = {X 217.0370, Y 8.1868, Z -2.1667, A 0.000, B 0.000, C 0.000 }
gfCNCPoint2[405] = {X 223.4805, Y 8.1868, Z -2.1667, A 0.000, B 0.000, C 0.000 }
gfCNCPoint2[406] = {X 224.3706, Y 8.2871, Z -2.1667, A 0.000, B 0.000, C 0.000 }
gfCNCPoint2[407] = {X 225.2160, Y 8.5829, Z -2.1667, A 0.000, B 0.000, C 0.000 }
gfCNCPoint2[408] = {X 225.9744, Y 9.0595, Z -2.1667, A 0.000, B 0.000, C 0.000 }
gfCNCPoint2[409] = {X 226.6078, Y 9.6929, Z -2.1667, A 0.000, B 0.000, C 0.000 }
gfCNCPoint2[410] = {X 227.0844, Y 10.4513, Z -2.1667, A 0.000, B 0.000, C 0.000 }
gfCNCPoint2[411] = {X 227.3802, Y 11.2967, Z -2.1667, A 0.000, B 0.000, C 0.000 }
gfCNCPoint2[412] = {X 227.4805, Y 12.1868, Z -2.1667, A 0.000, B 0.000, C 0.000 }
gfCNCPoint2[413] = {X 227.4803, Y 13.0192, Z -2.1667, A 0.000, B 0.000, C 0.000 }
gfCNCPoint2[414] = {X 227.3716, Y 13.9050, Z -2.1667, A 0.000, B 0.000, C 0.000 }
gfCNCPoint2[415] = {X 227.0692, Y 14.7447, Z -2.1667, A 0.000, B 0.000, C 0.000 }
gfCNCPoint2[416] = {X 226.5881, Y 15.4965, Z -2.1667, A 0.000, B 0.000, C 0.000 }
gfCNCPoint2[417] = {X 225.9523, Y 16.1229, Z -2.1667, A 0.000, B 0.000, C 0.000 }
gfCNCPoint2[418] = {X 225.9532, Y 41.0668, Z -2.1667, A 0.000, B 0.000, C 0.000 }
gfCNCPoint2[419] = {X 226.0921, Y 41.1790, Z -2.1667, A 0.000, B 0.000, C 0.000 }
gfCNCPoint2[420] = {X 226.6780, Y 41.8055, Z -2.1667, A 0.000, B 0.000, C 0.000 }
gfCNCPoint2[421] = {X 227.1169, Y 42.5425, Z -2.1667, A 0.000, B 0.000, C 0.000 }
gfCNCPoint2[422] = {X 227.3885, Y 43.3561, Z -2.1667, A 0.000, B 0.000, C 0.000 }
gfCNCPoint2[423] = {X 227.4805, Y 44.2089, Z -2.1667, A 0.000, B 0.000, C 0.000 }
gfCNCPoint2[424] = {X 227.4805, Y 45.0000, Z -2.1667, A 0.000, B 0.000, C 0.000 }
gfCNCPoint2[425] = {X 227.3802, Y 45.8901, Z -2.1667, A 0.000, B 0.000, C 0.000 }
gfCNCPoint2[426] = {X 227.0844, Y 46.7355, Z -2.1667, A 0.000, B 0.000, C 0.000 }
gfCNCPoint2[427] = {X 226.6078, Y 47.4940, Z -2.1667, A 0.000, B 0.000, C 0.000 }
gfCNCPoint2[428] = {X 225.9744, Y 48.1273, Z -2.1667, A 0.000, B 0.000, C 0.000 }
gfCNCPoint2[429] = {X 225.2160, Y 48.6039, Z -2.1667, A 0.000, B 0.000, C 0.000 }
gfCNCPoint2[430] = {X 224.3706, Y 48.8997, Z -2.1667, A 0.000, B 0.000, C 0.000 }
gfCNCPoint2[431] = {X 223.4805, Y 49.0000, Z -2.1667, A 0.000, B 0.000, C 0.000 }
gfCNCPoint2[432] = {X 217.0370, Y 49.0000, Z -2.1667, A 0.000, B 0.000, C 0.000 }
gfCNCPoint2[433] = {X 216.1469, Y 48.8997, Z -2.1667, A 0.000, B 0.000, C 0.000 }
gfCNCPoint2[434] = {X 215.3015, Y 48.6039, Z -2.1667, A 0.000, B 0.000, C 0.000 }
gfCNCPoint2[435] = {X 214.5430, Y 48.1273, Z -2.1667, A 0.000, B 0.000, C 0.000 }
gfCNCPoint2[436] = {X 213.9097, Y 47.4939, Z -2.1667, A 0.000, B 0.000, C 0.000 }
gfCNCPoint2[437] = {X 213.4331, Y 46.7355, Z -2.1667, A 0.000, B 0.000, C 0.000 }
gfCNCPoint2[438] = {X 213.1373, Y 45.8900, Z -2.1667, A 0.000, B 0.000, C 0.000 }
gfCNCPoint2[439] = {X 213.0370, Y 45.0000, Z -2.1667, A 0.000, B 0.000, C 0.000 }
gfCNCPoint2[440] = {X 213.0370, Y 44.1994, Z -2.1667, A 0.000, B 0.000, C 0.000 }
gfCNCPoint2[441] = {X 213.1550, Y 43.2426, Z -2.1667, A 0.000, B 0.000, C 0.000 }
gfCNCPoint2[442] = {X 213.5021, Y 42.3431, Z -2.1667, A 0.000, B 0.000, C 0.000 }
gfCNCPoint2[443] = {X 214.0573, Y 41.5550, Z -2.1667, A 0.000, B 0.000, C 0.000 }
gfCNCPoint2[444] = {X 214.5605, Y 40.9999, Z -2.1667, A 0.000, B 0.000, C 0.000 }
gfCNCPoint2[445] = {X 214.5659, Y 40.3075, Z -2.1667, A 0.000, B 0.000, C 0.000 }
gfCNCPoint2[446] = {X 214.5659, Y 28.5742, Z -2.1667, A 0.000, B 0.000, C 0.000 }
gfCNCPoint2[447] = {X 210.4859, Y 28.5742, Z -2.1667, A 0.000, B 0.000, C 0.000 }
gfCNCPoint2[448] = {X 210.4859, Y 28.5742, Z 0.8333, A 0.000, B 0.000, C 0.000 }
gfCNCPoint2[449] = {X 210.4859, Y 28.5742, Z 11.0000, A 0.000, B 0.000, C 0.000 }
gfCNCPoint2[450] = {X 273.6030, Y 28.5937, Z 11.0000, A 0.000, B 0.000, C 0.000 }
gfCNCPoint2[451] = {X 273.6030, Y 28.5937, Z 0.8333, A 0.000, B 0.000, C 0.000 }
gfCNCPoint2[452] = {X 273.6030, Y 28.5937, Z -2.1667, A 0.000, B 0.000, C 0.000 }
gfCNCPoint2[453] = {X 269.5230, Y 28.5936, Z -2.1667, A 0.000, B 0.000, C 0.000 }
gfCNCPoint2[454] = {X 269.5229, Y 40.9128, Z -2.1667, A 0.000, B 0.000, C 0.000 }
gfCNCPoint2[455] = {X 269.5368, Y 40.9240, Z -2.1667, A 0.000, B 0.000, C 0.000 }
gfCNCPoint2[456] = {X 270.1695, Y 41.5935, Z -2.1667, A 0.000, B 0.000, C 0.000 }
gfCNCPoint2[457] = {X 270.6458, Y 42.3820, Z -2.1667, A 0.000, B 0.000, C 0.000 }
gfCNCPoint2[458] = {X 270.9441, Y 43.2536, Z -2.1667, A 0.000, B 0.000, C 0.000 }
gfCNCPoint2[459] = {X 271.0508, Y 44.1686, Z -2.1667, A 0.000, B 0.000, C 0.000 }
gfCNCPoint2[460] = {X 271.0510, Y 45.0000, Z -2.1667, A 0.000, B 0.000, C 0.000 }
gfCNCPoint2[461] = {X 270.9427, Y 45.9613, Z -2.1667, A 0.000, B 0.000, C 0.000 }
gfCNCPoint2[462] = {X 270.6232, Y 46.8744, Z -2.1667, A 0.000, B 0.000, C 0.000 }
gfCNCPoint2[463] = {X 270.1085, Y 47.6935, Z -2.1667, A 0.000, B 0.000, C 0.000 }
gfCNCPoint2[464] = {X 269.4245, Y 48.3775, Z -2.1667, A 0.000, B 0.000, C 0.000 }
gfCNCPoint2[465] = {X 268.6054, Y 48.8922, Z -2.1667, A 0.000, B 0.000, C 0.000 }
gfCNCPoint2[466] = {X 267.6923, Y 49.2117, Z -2.1667, A 0.000, B 0.000, C 0.000 }
gfCNCPoint2[467] = {X 266.7310, Y 49.3200, Z -2.1667, A 0.000, B 0.000, C 0.000 }
gfCNCPoint2[468] = {X 260.2876, Y 49.3200, Z -2.1667, A 0.000, B 0.000, C 0.000 }
gfCNCPoint2[469] = {X 259.3310, Y 49.2128, Z -2.1667, A 0.000, B 0.000, C 0.000 }
gfCNCPoint2[470] = {X 258.4219, Y 48.8963, Z -2.1667, A 0.000, B 0.000, C 0.000 }
gfCNCPoint2[471] = {X 257.6054, Y 48.3865, Z -2.1667, A 0.000, B 0.000, C 0.000 }
gfCNCPoint2[472] = {X 256.9221, Y 47.7085, Z -2.1667, A 0.000, B 0.000, C 0.000 }
gfCNCPoint2[473] = {X 256.4059, Y 46.8960, Z -2.1667, A 0.000, B 0.000, C 0.000 }
gfCNCPoint2[474] = {X 256.0824, Y 45.9894, Z -2.1667, A 0.000, B 0.000, C 0.000 }
gfCNCPoint2[475] = {X 255.9677, Y 45.0336, Z -2.1667, A 0.000, B 0.000, C 0.000 }
gfCNCPoint2[476] = {X 255.9680, Y 44.1494, Z -2.1667, A 0.000, B 0.000, C 0.000 }
gfCNCPoint2[477] = {X 256.0784, Y 43.2364, Z -2.1667, A 0.000, B 0.000, C 0.000 }
gfCNCPoint2[478] = {X 256.3796, Y 42.3675, Z -2.1667, A 0.000, B 0.000, C 0.000 }
gfCNCPoint2[479] = {X 256.8579, Y 41.5821, Z -2.1667, A 0.000, B 0.000, C 0.000 }
gfCNCPoint2[480] = {X 257.4915, Y 40.9157, Z -2.1667, A 0.000, B 0.000, C 0.000 }
gfCNCPoint2[481] = {X 257.4915, Y 34.4738, Z -2.1667, A 0.000, B 0.000, C 0.000 }
gfCNCPoint2[482] = {X 254.7668, Y 34.4738, Z -2.1667, A 0.000, B 0.000, C 0.000 }
gfCNCPoint2[483] = {X 250.4836, Y 42.8180, Z -2.1667, A 0.000, B 0.000, C 0.000 }
gfCNCPoint2[484] = {X 250.6527, Y 43.4860, Z -2.1667, A 0.000, B 0.000, C 0.000 }
gfCNCPoint2[485] = {X 250.7134, Y 44.1723, Z -2.1667, A 0.000, B 0.000, C 0.000 }
gfCNCPoint2[486] = {X 250.7136, Y 45.0000, Z -2.1667, A 0.000, B 0.000, C 0.000 }
gfCNCPoint2[487] = {X 250.6052, Y 45.9613, Z -2.1667, A 0.000, B 0.000, C 0.000 }
gfCNCPoint2[488] = {X 250.2857, Y 46.8744, Z -2.1667, A 0.000, B 0.000, C 0.000 }
gfCNCPoint2[489] = {X 249.7711, Y 47.6935, Z -2.1667, A 0.000, B 0.000, C 0.000 }
gfCNCPoint2[490] = {X 249.0870, Y 48.3775, Z -2.1667, A 0.000, B 0.000, C 0.000 }
gfCNCPoint2[491] = {X 248.2679, Y 48.8922, Z -2.1667, A 0.000, B 0.000, C 0.000 }
gfCNCPoint2[492] = {X 247.3548, Y 49.2117, Z -2.1667, A 0.000, B 0.000, C 0.000 }
gfCNCPoint2[493] = {X 246.3936, Y 49.3200, Z -2.1667, A 0.000, B 0.000, C 0.000 }
gfCNCPoint2[494] = {X 239.8075, Y 49.3200, Z -2.1667, A 0.000, B 0.000, C 0.000 }
gfCNCPoint2[495] = {X 238.8462, Y 49.2117, Z -2.1667, A 0.000, B 0.000, C 0.000 }
gfCNCPoint2[496] = {X 237.9331, Y 48.8922, Z -2.1667, A 0.000, B 0.000, C 0.000 }
gfCNCPoint2[497] = {X 237.1141, Y 48.3775, Z -2.1667, A 0.000, B 0.000, C 0.000 }
gfCNCPoint2[498] = {X 236.4300, Y 47.6935, Z -2.1667, A 0.000, B 0.000, C 0.000 }
gfCNCPoint2[499] = {X 235.9153, Y 46.8745, Z -2.1667, A 0.000, B 0.000, C 0.000 }
gfCNCPoint2[500] = {X 235.5958, Y 45.9614, Z -2.1667, A 0.000, B 0.000, C 0.000 }
gfCNCPoint2[501] = {X 235.4875, Y 45.0001, Z -2.1667, A 0.000, B 0.000, C 0.000 }
gfCNCPoint2[502] = {X 235.4879, Y 44.1494, Z -2.1667, A 0.000, B 0.000, C 0.000 }
gfCNCPoint2[503] = {X 235.5856, Y 43.2935, Z -2.1667, A 0.000, B 0.000, C 0.000 }
gfCNCPoint2[504] = {X 235.8511, Y 42.4740, Z -2.1667, A 0.000, B 0.000, C 0.000 }
gfCNCPoint2[505] = {X 236.2739, Y 41.7236, Z -2.1667, A 0.000, B 0.000, C 0.000 }
gfCNCPoint2[506] = {X 236.8373, Y 41.0719, Z -2.1667, A 0.000, B 0.000, C 0.000 }
gfCNCPoint2[507] = {X 237.5187, Y 40.5449, Z -2.1667, A 0.000, B 0.000, C 0.000 }
gfCNCPoint2[508] = {X 238.2911, Y 40.1637, Z -2.1667, A 0.000, B 0.000, C 0.000 }
gfCNCPoint2[509] = {X 242.2807, Y 32.3546, Z -2.1667, A 0.000, B 0.000, C 0.000 }
gfCNCPoint2[510] = {X 241.1108, Y 31.5683, Z -2.1667, A 0.000, B 0.000, C 0.000 }
gfCNCPoint2[511] = {X 240.0477, Y 30.6426, Z -2.1667, A 0.000, B 0.000, C 0.000 }
gfCNCPoint2[512] = {X 239.1080, Y 29.5920, Z -2.1667, A 0.000, B 0.000, C 0.000 }
gfCNCPoint2[513] = {X 238.3062, Y 28.4327, Z -2.1667, A 0.000, B 0.000, C 0.000 }
gfCNCPoint2[514] = {X 237.6547, Y 27.1827, Z -2.1667, A 0.000, B 0.000, C 0.000 }
gfCNCPoint2[515] = {X 237.1636, Y 25.8615, Z -2.1667, A 0.000, B 0.000, C 0.000 }
gfCNCPoint2[516] = {X 236.7434, Y 24.0500, Z -2.1667, A 0.000, B 0.000, C 0.000 }
gfCNCPoint2[517] = {X 236.5293, Y 22.2028, Z -2.1667, A 0.000, B 0.000, C 0.000 }
gfCNCPoint2[518] = {X 236.5240, Y 20.3432, Z -2.1667, A 0.000, B 0.000, C 0.000 }
gfCNCPoint2[519] = {X 236.7274, Y 18.4948, Z -2.1667, A 0.000, B 0.000, C 0.000 }
gfCNCPoint2[520] = {X 237.1372, Y 16.6810, Z -2.1667, A 0.000, B 0.000, C 0.000 }
gfCNCPoint2[521] = {X 237.7074, Y 15.1054, Z -2.1667, A 0.000, B 0.000, C 0.000 }
gfCNCPoint2[522] = {X 238.4943, Y 13.6261, Z -2.1667, A 0.000, B 0.000, C 0.000 }
gfCNCPoint2[523] = {X 239.4820, Y 12.2726, Z -2.1667, A 0.000, B 0.000, C 0.000 }
gfCNCPoint2[524] = {X 240.6508, Y 11.0720, Z -2.1667, A 0.000, B 0.000, C 0.000 }
gfCNCPoint2[525] = {X 241.9774, Y 10.0483, Z -2.1667, A 0.000, B 0.000, C 0.000 }
gfCNCPoint2[526] = {X 243.4350, Y 9.2220, Z -2.1667, A 0.000, B 0.000, C 0.000 }
gfCNCPoint2[527] = {X 244.9947, Y 8.6097, Z -2.1667, A 0.000, B 0.000, C 0.000 }
gfCNCPoint2[528] = {X 246.6252, Y 8.2236, Z -2.1667, A 0.000, B 0.000, C 0.000 }
gfCNCPoint2[529] = {X 248.7221, Y 7.9518, Z -2.1667, A 0.000, B 0.000, C 0.000 }
gfCNCPoint2[530] = {X 250.8350, Y 7.8716, Z -2.1667, A 0.000, B 0.000, C 0.000 }
gfCNCPoint2[531] = {X 266.7634, Y 7.8716, Z -2.1667, A 0.000, B 0.000, C 0.000 }
gfCNCPoint2[532] = {X 267.7184, Y 7.9863, Z -2.1667, A 0.000, B 0.000, C 0.000 }
gfCNCPoint2[533] = {X 268.6244, Y 8.3095, Z -2.1667, A 0.000, B 0.000, C 0.000 }
gfCNCPoint2[534] = {X 269.4365, Y 8.8249, Z -2.1667, A 0.000, B 0.000, C 0.000 }
gfCNCPoint2[535] = {X 270.1145, Y 9.5072, Z -2.1667, A 0.000, B 0.000, C 0.000 }
gfCNCPoint2[536] = {X 270.6249, Y 10.3226, Z -2.1667, A 0.000, B 0.000, C 0.000 }
gfCNCPoint2[537] = {X 270.9423, Y 11.2306, Z -2.1667, A 0.000, B 0.000, C 0.000 }
gfCNCPoint2[538] = {X 271.0510, Y 12.1863, Z -2.1667, A 0.000, B 0.000, C 0.000 }
gfCNCPoint2[539] = {X 271.0508, Y 13.0225, Z -2.1667, A 0.000, B 0.000, C 0.000 }
gfCNCPoint2[540] = {X 270.9424, Y 13.9407, Z -2.1667, A 0.000, B 0.000, C 0.000 }
gfCNCPoint2[541] = {X 270.6411, Y 14.8148, Z -2.1667, A 0.000, B 0.000, C 0.000 }
gfCNCPoint2[542] = {X 270.1607, Y 15.6048, Z -2.1667, A 0.000, B 0.000, C 0.000 }
gfCNCPoint2[543] = {X 269.5231, Y 16.2745, Z -2.1667, A 0.000, B 0.000, C 0.000 }
gfCNCPoint2[544] = {X 269.5230, Y 28.5936, Z -2.1667, A 0.000, B 0.000, C 0.000 }
gfCNCPoint2[545] = {X 273.5230, Y 28.5937, Z -2.1667, A 0.000, B 0.000, C 0.000 }
gfCNCPoint2[546] = {X 269.4430, Y 28.5936, Z -2.1667, A 0.000, B 0.000, C 0.000 }
gfCNCPoint2[547] = {X 269.4429, Y 40.9512, Z -2.1667, A 0.000, B 0.000, C 0.000 }
gfCNCPoint2[548] = {X 269.4857, Y 40.9856, Z -2.1667, A 0.000, B 0.000, C 0.000 }
gfCNCPoint2[549] = {X 270.1063, Y 41.6427, Z -2.1667, A 0.000, B 0.000, C 0.000 }
gfCNCPoint2[550] = {X 270.5735, Y 42.4164, Z -2.1667, A 0.000, B 0.000, C 0.000 }
gfCNCPoint2[551] = {X 270.8661, Y 43.2715, Z -2.1667, A 0.000, B 0.000, C 0.000 }
gfCNCPoint2[552] = {X 270.9708, Y 44.1693, Z -2.1667, A 0.000, B 0.000, C 0.000 }
gfCNCPoint2[553] = {X 270.9710, Y 45.0000, Z -2.1667, A 0.000, B 0.000, C 0.000 }
gfCNCPoint2[554] = {X 270.8647, Y 45.9435, Z -2.1667, A 0.000, B 0.000, C 0.000 }
gfCNCPoint2[555] = {X 270.5511, Y 46.8397, Z -2.1667, A 0.000, B 0.000, C 0.000 }
gfCNCPoint2[556] = {X 270.0460, Y 47.6436, Z -2.1667, A 0.000, B 0.000, C 0.000 }
gfCNCPoint2[557] = {X 269.3746, Y 48.3150, Z -2.1667, A 0.000, B 0.000, C 0.000 }
gfCNCPoint2[558] = {X 268.5707, Y 48.8201, Z -2.1667, A 0.000, B 0.000, C 0.000 }
gfCNCPoint2[559] = {X 267.6745, Y 49.1337, Z -2.1667, A 0.000, B 0.000, C 0.000 }
gfCNCPoint2[560] = {X 266.7310, Y 49.2400, Z -2.1667, A 0.000, B 0.000, C 0.000 }
gfCNCPoint2[561] = {X 260.2876, Y 49.2400, Z -2.1667, A 0.000, B 0.000, C 0.000 }
gfCNCPoint2[562] = {X 259.3487, Y 49.1347, Z -2.1667, A 0.000, B 0.000, C 0.000 }
gfCNCPoint2[563] = {X 258.4564, Y 48.8242, Z -2.1667, A 0.000, B 0.000, C 0.000 }
gfCNCPoint2[564] = {X 257.6550, Y 48.3238, Z -2.1667, A 0.000, B 0.000, C 0.000 }
gfCNCPoint2[565] = {X 256.9844, Y 47.6583, Z -2.1667, A 0.000, B 0.000, C 0.000 }
gfCNCPoint2[566] = {X 256.4777, Y 46.8609, Z -2.1667, A 0.000, B 0.000, C 0.000 }
gfCNCPoint2[567] = {X 256.1603, Y 45.9711, Z -2.1667, A 0.000, B 0.000, C 0.000 }
gfCNCPoint2[568] = {X 256.0477, Y 45.0330, Z -2.1667, A 0.000, B 0.000, C 0.000 }
gfCNCPoint2[569] = {X 256.0480, Y 44.1505, Z -2.1667, A 0.000, B 0.000, C 0.000 }
gfCNCPoint2[570] = {X 256.1585, Y 43.2454, Z -2.1667, A 0.000, B 0.000, C 0.000 }
gfCNCPoint2[571] = {X 256.4599, Y 42.3850, Z -2.1667, A 0.000, B 0.000, C 0.000 }
gfCNCPoint2[572] = {X 256.9383, Y 41.6088, Z -2.1667, A 0.000, B 0.000, C 0.000 }
gfCNCPoint2[573] = {X 257.5715, Y 40.9529, Z -2.1667, A 0.000, B 0.000, C 0.000 }
gfCNCPoint2[574] = {X 257.5715, Y 34.3938, Z -2.1667, A 0.000, B 0.000, C 0.000 }
gfCNCPoint2[575] = {X 254.7179, Y 34.3938, Z -2.1667, A 0.000, B 0.000, C 0.000 }
gfCNCPoint2[576] = {X 250.3968, Y 42.8118, Z -2.1667, A 0.000, B 0.000, C 0.000 }
gfCNCPoint2[577] = {X 250.5709, Y 43.4827, Z -2.1667, A 0.000, B 0.000, C 0.000 }
gfCNCPoint2[578] = {X 250.6334, Y 44.1730, Z -2.1667, A 0.000, B 0.000, C 0.000 }
gfCNCPoint2[579] = {X 250.6336, Y 45.0000, Z -2.1667, A 0.000, B 0.000, C 0.000 }
gfCNCPoint2[580] = {X 250.5273, Y 45.9435, Z -2.1667, A 0.000, B 0.000, C 0.000 }
gfCNCPoint2[581] = {X 250.2137, Y 46.8397, Z -2.1667, A 0.000, B 0.000, C 0.000 }
gfCNCPoint2[582] = {X 249.7085, Y 47.6436, Z -2.1667, A 0.000, B 0.000, C 0.000 }
gfCNCPoint2[583] = {X 249.0372, Y 48.3150, Z -2.1667, A 0.000, B 0.000, C 0.000 }
gfCNCPoint2[584] = {X 248.2332, Y 48.8201, Z -2.1667, A 0.000, B 0.000, C 0.000 }
gfCNCPoint2[585] = {X 247.3370, Y 49.1337, Z -2.1667, A 0.000, B 0.000, C 0.000 }
gfCNCPoint2[586] = {X 246.3936, Y 49.2400, Z -2.1667, A 0.000, B 0.000, C 0.000 }
gfCNCPoint2[587] = {X 239.8075, Y 49.2400, Z -2.1667, A 0.000, B 0.000, C 0.000 }
gfCNCPoint2[588] = {X 238.8640, Y 49.1337, Z -2.1667, A 0.000, B 0.000, C 0.000 }
gfCNCPoint2[589] = {X 237.9679, Y 48.8201, Z -2.1667, A 0.000, B 0.000, C 0.000 }
gfCNCPoint2[590] = {X 237.1639, Y 48.3150, Z -2.1667, A 0.000, B 0.000, C 0.000 }
gfCNCPoint2[591] = {X 236.4926, Y 47.6436, Z -2.1667, A 0.000, B 0.000, C 0.000 }
gfCNCPoint2[592] = {X 235.9874, Y 46.8397, Z -2.1667, A 0.000, B 0.000, C 0.000 }
gfCNCPoint2[593] = {X 235.6738, Y 45.9436, Z -2.1667, A 0.000, B 0.000, C 0.000 }
gfCNCPoint2[594] = {X 235.5675, Y 45.0001, Z -2.1667, A 0.000, B 0.000, C 0.000 }
gfCNCPoint2[595] = {X 235.5679, Y 44.1505, Z -2.1667, A 0.000, B 0.000, C 0.000 }
gfCNCPoint2[596] = {X 235.6649, Y 43.3054, Z -2.1667, A 0.000, B 0.000, C 0.000 }
gfCNCPoint2[597] = {X 235.9285, Y 42.4967, Z -2.1667, A 0.000, B 0.000, C 0.000 }
gfCNCPoint2[598] = {X 236.3483, Y 41.7570, Z -2.1667, A 0.000, B 0.000, C 0.000 }
gfCNCPoint2[599] = {X 236.9073, Y 41.1159, Z -2.1667, A 0.000, B 0.000, C 0.000 }
gfCNCPoint2[600] = {X 237.5830, Y 40.5992, Z -2.1667, A 0.000, B 0.000, C 0.000 }
gfCNCPoint2[601] = {X 238.3482, Y 40.2278, Z -2.1667, A 0.000, B 0.000, C 0.000 }
gfCNCPoint2[602] = {X 242.3864, Y 32.3235, Z -2.1667, A 0.000, B 0.000, C 0.000 }
gfCNCPoint2[603] = {X 241.2095, Y 31.5430, Z -2.1667, A 0.000, B 0.000, C 0.000 }
gfCNCPoint2[604] = {X 240.1398, Y 30.6210, Z -2.1667, A 0.000, B 0.000, C 0.000 }
gfCNCPoint2[605] = {X 239.1943, Y 29.5721, Z -2.1667, A 0.000, B 0.000, C 0.000 }
gfCNCPoint2[606] = {X 238.3877, Y 28.4129, Z -2.1667, A 0.000, B 0.000, C 0.000 }
gfCNCPoint2[607] = {X 237.7329, Y 27.1618, Z -2.1667, A 0.000, B 0.000, C 0.000 }
gfCNCPoint2[608] = {X 237.2402, Y 25.8383, Z -2.1667, A 0.000, B 0.000, C 0.000 }
gfCNCPoint2[609] = {X 236.8221, Y 24.0357, Z -2.1667, A 0.000, B 0.000, C 0.000 }
gfCNCPoint2[610] = {X 236.6091, Y 22.1976, Z -2.1667, A 0.000, B 0.000, C 0.000 }
gfCNCPoint2[611] = {X 236.6039, Y 20.3472, Z -2.1667, A 0.000, B 0.000, C 0.000 }
gfCNCPoint2[612] = {X 236.8064, Y 18.5078, Z -2.1667, A 0.000, B 0.000, C 0.000 }
gfCNCPoint2[613] = {X 237.2141, Y 16.7029, Z -2.1667, A 0.000, B 0.000, C 0.000 }
gfCNCPoint2[614] = {X 237.7805, Y 15.1379, Z -2.1667, A 0.000, B 0.000, C 0.000 }
gfCNCPoint2[615] = {X 238.5621, Y 13.6685, Z -2.1667, A 0.000, B 0.000, C 0.000 }
gfCNCPoint2[616] = {X 239.5432, Y 12.3241, Z -2.1667, A 0.000, B 0.000, C 0.000 }
gfCNCPoint2[617] = {X 240.7042, Y 11.1316, Z -2.1667, A 0.000, B 0.000, C 0.000 }
gfCNCPoint2[618] = {X 242.0219, Y 10.1148, Z -2.1667, A 0.000, B 0.000, C 0.000 }
gfCNCPoint2[619] = {X 243.4698, Y 9.2941, Z -2.1667, A 0.000, B 0.000, C 0.000 }
gfCNCPoint2[620] = {X 245.0190, Y 8.6859, Z -2.1667, A 0.000, B 0.000, C 0.000 }
gfCNCPoint2[621] = {X 246.6386, Y 8.3025, Z -2.1667, A 0.000, B 0.000, C 0.000 }
gfCNCPoint2[622] = {X 248.7287, Y 8.0316, Z -2.1667, A 0.000, B 0.000, C 0.000 }
gfCNCPoint2[623] = {X 250.8347, Y 7.9516, Z -2.1667, A 0.000, B 0.000, C 0.000 }
gfCNCPoint2[624] = {X 266.7627, Y 7.9516, Z -2.1667, A 0.000, B 0.000, C 0.000 }
gfCNCPoint2[625] = {X 267.7001, Y 8.0642, Z -2.1667, A 0.000, B 0.000, C 0.000 }
gfCNCPoint2[626] = {X 268.5893, Y 8.3813, Z -2.1667, A 0.000, B 0.000, C 0.000 }
gfCNCPoint2[627] = {X 269.3864, Y 8.8873, Z -2.1667, A 0.000, B 0.000, C 0.000 }
gfCNCPoint2[628] = {X 270.0519, Y 9.5569, Z -2.1667, A 0.000, B 0.000, C 0.000 }
gfCNCPoint2[629] = {X 270.5528, Y 10.3572, Z -2.1667, A 0.000, B 0.000, C 0.000 }
gfCNCPoint2[630] = {X 270.8643, Y 11.2484, Z -2.1667, A 0.000, B 0.000, C 0.000 }
gfCNCPoint2[631] = {X 270.9710, Y 12.1865, Z -2.1667, A 0.000, B 0.000, C 0.000 }
gfCNCPoint2[632] = {X 270.9708, Y 13.0217, Z -2.1667, A 0.000, B 0.000, C 0.000 }
gfCNCPoint2[633] = {X 270.8623, Y 13.9319, Z -2.1667, A 0.000, B 0.000, C 0.000 }
gfCNCPoint2[634] = {X 270.5608, Y 14.7975, Z -2.1667, A 0.000, B 0.000, C 0.000 }
gfCNCPoint2[635] = {X 270.0802, Y 15.5781, Z -2.1667, A 0.000, B 0.000, C 0.000 }
gfCNCPoint2[636] = {X 269.4431, Y 16.2372, Z -2.1667, A 0.000, B 0.000, C 0.000 }
gfCNCPoint2[637] = {X 269.4430, Y 28.5936, Z -2.1667, A 0.000, B 0.000, C 0.000 }
gfCNCPoint2[638] = {X 273.4430, Y 28.5937, Z -2.1667, A 0.000, B 0.000, C 0.000 }
gfCNCPoint2[639] = {X 269.3630, Y 28.5936, Z -2.1667, A 0.000, B 0.000, C 0.000 }
gfCNCPoint2[640] = {X 269.3629, Y 40.9895, Z -2.1667, A 0.000, B 0.000, C 0.000 }
gfCNCPoint2[641] = {X 269.4347, Y 41.0472, Z -2.1667, A 0.000, B 0.000, C 0.000 }
gfCNCPoint2[642] = {X 270.0432, Y 41.6918, Z -2.1667, A 0.000, B 0.000, C 0.000 }
gfCNCPoint2[643] = {X 270.5013, Y 42.4507, Z -2.1667, A 0.000, B 0.000, C 0.000 }
gfCNCPoint2[644] = {X 270.7882, Y 43.2895, Z -2.1667, A 0.000, B 0.000, C 0.000 }
gfCNCPoint2[645] = {X 270.8909, Y 44.1700, Z -2.1667, A 0.000, B 0.000, C 0.000 }
gfCNCPoint2[646] = {X 270.8910, Y 45.0000, Z -2.1667, A 0.000, B 0.000, C 0.000 }
gfCNCPoint2[647] = {X 270.7867, Y 45.9257, Z -2.1667, A 0.000, B 0.000, C 0.000 }
gfCNCPoint2[648] = {X 270.4791, Y 46.8050, Z -2.1667, A 0.000, B 0.000, C 0.000 }
gfCNCPoint2[649] = {X 269.9835, Y 47.5937, Z -2.1667, A 0.000, B 0.000, C 0.000 }
gfCNCPoint2[650] = {X 269.3247, Y 48.2524, Z -2.1667, A 0.000, B 0.000, C 0.000 }
gfCNCPoint2[651] = {X 268.5360, Y 48.7480, Z -2.1667, A 0.000, B 0.000, C 0.000 }
gfCNCPoint2[652] = {X 267.6567, Y 49.0557, Z -2.1667, A 0.000, B 0.000, C 0.000 }
gfCNCPoint2[653] = {X 266.7310, Y 49.1600, Z -2.1667, A 0.000, B 0.000, C 0.000 }
gfCNCPoint2[654] = {X 260.2876, Y 49.1600, Z -2.1667, A 0.000, B 0.000, C 0.000 }
gfCNCPoint2[655] = {X 259.3664, Y 49.0567, Z -2.1667, A 0.000, B 0.000, C 0.000 }
gfCNCPoint2[656] = {X 258.4910, Y 48.7520, Z -2.1667, A 0.000, B 0.000, C 0.000 }
gfCNCPoint2[657] = {X 257.7047, Y 48.2611, Z -2.1667, A 0.000, B 0.000, C 0.000 }
gfCNCPoint2[658] = {X 257.0467, Y 47.6082, Z -2.1667, A 0.000, B 0.000, C 0.000 }
gfCNCPoint2[659] = {X 256.5496, Y 46.8258, Z -2.1667, A 0.000, B 0.000, C 0.000 }
gfCNCPoint2[660] = {X 256.2381, Y 45.9527, Z -2.1667, A 0.000, B 0.000, C 0.000 }
gfCNCPoint2[661] = {X 256.1277, Y 45.0324, Z -2.1667, A 0.000, B 0.000, C 0.000 }
gfCNCPoint2[662] = {X 256.1280, Y 44.1516, Z -2.1667, A 0.000, B 0.000, C 0.000 }
gfCNCPoint2[663] = {X 256.2385, Y 43.2545, Z -2.1667, A 0.000, B 0.000, C 0.000 }
gfCNCPoint2[664] = {X 256.5401, Y 42.4026, Z -2.1667, A 0.000, B 0.000, C 0.000 }
gfCNCPoint2[665] = {X 257.0187, Y 41.6358, Z -2.1667, A 0.000, B 0.000, C 0.000 }
gfCNCPoint2[666] = {X 257.6515, Y 40.9906, Z -2.1667, A 0.000, B 0.000, C 0.000 }
gfCNCPoint2[667] = {X 257.6515, Y 34.3138, Z -2.1667, A 0.000, B 0.000, C 0.000 }
gfCNCPoint2[668] = {X 254.6690, Y 34.3138, Z -2.1667, A 0.000, B 0.000, C 0.000 }
gfCNCPoint2[669] = {X 250.3099, Y 42.8060, Z -2.1667, A 0.000, B 0.000, C 0.000 }
gfCNCPoint2[670] = {X 250.4891, Y 43.4796, Z -2.1667, A 0.000, B 0.000, C 0.000 }
gfCNCPoint2[671] = {X 250.5534, Y 44.1736, Z -2.1667, A 0.000, B 0.000, C 0.000 }
gfCNCPoint2[672] = {X 250.5536, Y 45.0000, Z -2.1667, A 0.000, B 0.000, C 0.000 }
gfCNCPoint2[673] = {X 250.4493, Y 45.9257, Z -2.1667, A 0.000, B 0.000, C 0.000 }
gfCNCPoint2[674] = {X 250.1416, Y 46.8050, Z -2.1667, A 0.000, B 0.000, C 0.000 }
gfCNCPoint2[675] = {X 249.6460, Y 47.5937, Z -2.1667, A 0.000, B 0.000, C 0.000 }
gfCNCPoint2[676] = {X 248.9873, Y 48.2524, Z -2.1667, A 0.000, B 0.000, C 0.000 }
gfCNCPoint2[677] = {X 248.1985, Y 48.7480, Z -2.1667, A 0.000, B 0.000, C 0.000 }
gfCNCPoint2[678] = {X 247.3192, Y 49.0557, Z -2.1667, A 0.000, B 0.000, C 0.000 }
gfCNCPoint2[679] = {X 246.3936, Y 49.1600, Z -2.1667, A 0.000, B 0.000, C 0.000 }
gfCNCPoint2[680] = {X 239.8075, Y 49.1600, Z -2.1667, A 0.000, B 0.000, C 0.000 }
gfCNCPoint2[681] = {X 238.8818, Y 49.0557, Z -2.1667, A 0.000, B 0.000, C 0.000 }
gfCNCPoint2[682] = {X 238.0026, Y 48.7480, Z -2.1667, A 0.000, B 0.000, C 0.000 }
gfCNCPoint2[683] = {X 237.2138, Y 48.2524, Z -2.1667, A 0.000, B 0.000, C 0.000 }
gfCNCPoint2[684] = {X 236.5551, Y 47.5937, Z -2.1667, A 0.000, B 0.000, C 0.000 }
gfCNCPoint2[685] = {X 236.0595, Y 46.8050, Z -2.1667, A 0.000, B 0.000, C 0.000 }
gfCNCPoint2[686] = {X 235.7518, Y 45.9257, Z -2.1667, A 0.000, B 0.000, C 0.000 }
gfCNCPoint2[687] = {X 235.6475, Y 45.0000, Z -2.1667, A 0.000, B 0.000, C 0.000 }
gfCNCPoint2[688] = {X 235.6479, Y 44.1516, Z -2.1667, A 0.000, B 0.000, C 0.000 }
gfCNCPoint2[689] = {X 235.7441, Y 43.3174, Z -2.1667, A 0.000, B 0.000, C 0.000 }
gfCNCPoint2[690] = {X 236.0059, Y 42.5195, Z -2.1667, A 0.000, B 0.000, C 0.000 }
gfCNCPoint2[691] = {X 236.4226, Y 41.7905, Z -2.1667, A 0.000, B 0.000, C 0.000 }
gfCNCPoint2[692] = {X 236.9772, Y 41.1600, Z -2.1667, A 0.000, B 0.000, C 0.000 }
gfCNCPoint2[693] = {X 237.6471, Y 40.6537, Z -2.1667, A 0.000, B 0.000, C 0.000 }
gfCNCPoint2[694] = {X 238.4051, Y 40.2923, Z -2.1667, A 0.000, B 0.000, C 0.000 }
gfCNCPoint2[695] = {X 242.4924, Y 32.2919, Z -2.1667, A 0.000, B 0.000, C 0.000 }
gfCNCPoint2[696] = {X 241.3085, Y 31.5174, Z -2.1667, A 0.000, B 0.000, C 0.000 }
gfCNCPoint2[697] = {X 240.2321, Y 30.5992, Z -2.1667, A 0.000, B 0.000, C 0.000 }
gfCNCPoint2[698] = {X 239.2806, Y 29.5521, Z -2.1667, A 0.000, B 0.000, C 0.000 }
gfCNCPoint2[699] = {X 238.4693, Y 28.3931, Z -2.1667, A 0.000, B 0.000, C 0.000 }
gfCNCPoint2[700] = {X 237.8111, Y 27.1408, Z -2.1667, A 0.000, B 0.000, C 0.000 }
gfCNCPoint2[701] = {X 237.3168, Y 25.8152, Z -2.1667, A 0.000, B 0.000, C 0.000 }
gfCNCPoint2[702] = {X 236.9009, Y 24.0215, Z -2.1667, A 0.000, B 0.000, C 0.000 }
gfCNCPoint2[703] = {X 236.6890, Y 22.1924, Z -2.1667, A 0.000, B 0.000, C 0.000 }
gfCNCPoint2[704] = {X 236.6838, Y 20.3511, Z -2.1667, A 0.000, B 0.000, C 0.000 }
gfCNCPoint2[705] = {X 236.8853, Y 18.5209, Z -2.1667, A 0.000, B 0.000, C 0.000 }
gfCNCPoint2[706] = {X 237.2910, Y 16.7248, Z -2.1667, A 0.000, B 0.000, C 0.000 }
gfCNCPoint2[707] = {X 237.8536, Y 15.1704, Z -2.1667, A 0.000, B 0.000, C 0.000 }
gfCNCPoint2[708] = {X 238.6299, Y 13.7109, Z -2.1667, A 0.000, B 0.000, C 0.000 }
gfCNCPoint2[709] = {X 239.6044, Y 12.3756, Z -2.1667, A 0.000, B 0.000, C 0.000 }
gfCNCPoint2[710] = {X 240.7576, Y 11.1911, Z -2.1667, A 0.000, B 0.000, C 0.000 }
gfCNCPoint2[711] = {X 242.0664, Y 10.1813, Z -2.1667, A 0.000, B 0.000, C 0.000 }
gfCNCPoint2[712] = {X 243.5045, Y 9.3662, Z -2.1667, A 0.000, B 0.000, C 0.000 }
gfCNCPoint2[713] = {X 245.0433, Y 8.7622, Z -2.1667, A 0.000, B 0.000, C 0.000 }
gfCNCPoint2[714] = {X 246.6520, Y 8.3813, Z -2.1667, A 0.000, B 0.000, C 0.000 }
gfCNCPoint2[715] = {X 248.7352, Y 8.1113, Z -2.1667, A 0.000, B 0.000, C 0.000 }
gfCNCPoint2[716] = {X 250.8343, Y 8.0316, Z -2.1667, A 0.000, B 0.000, C 0.000 }
gfCNCPoint2[717] = {X 266.7621, Y 8.0316, Z -2.1667, A 0.000, B 0.000, C 0.000 }
gfCNCPoint2[718] = {X 267.6817, Y 8.1421, Z -2.1667, A 0.000, B 0.000, C 0.000 }
gfCNCPoint2[719] = {X 268.5542, Y 8.4532, Z -2.1667, A 0.000, B 0.000, C 0.000 }
gfCNCPoint2[720] = {X 269.3363, Y 8.9496, Z -2.1667, A 0.000, B 0.000, C 0.000 }
gfCNCPoint2[721] = {X 269.9892, Y 9.6067, Z -2.1667, A 0.000, B 0.000, C 0.000 }
gfCNCPoint2[722] = {X 270.4806, Y 10.3918, Z -2.1667, A 0.000, B 0.000, C 0.000 }
gfCNCPoint2[723] = {X 270.7863, Y 11.2662, Z -2.1667, A 0.000, B 0.000, C 0.000 }
gfCNCPoint2[724] = {X 270.8910, Y 12.1866, Z -2.1667, A 0.000, B 0.000, C 0.000 }
gfCNCPoint2[725] = {X 270.8908, Y 13.0208, Z -2.1667, A 0.000, B 0.000, C 0.000 }
gfCNCPoint2[726] = {X 270.7823, Y 13.9230, Z -2.1667, A 0.000, B 0.000, C 0.000 }
gfCNCPoint2[727] = {X 270.4805, Y 14.7800, Z -2.1667, A 0.000, B 0.000, C 0.000 }
gfCNCPoint2[728] = {X 269.9998, Y 15.5511, Z -2.1667, A 0.000, B 0.000, C 0.000 }
gfCNCPoint2[729] = {X 269.3631, Y 16.1995, Z -2.1667, A 0.000, B 0.000, C 0.000 }
gfCNCPoint2[730] = {X 269.3630, Y 28.5936, Z -2.1667, A 0.000, B 0.000, C 0.000 }
gfCNCPoint2[731] = {X 273.3630, Y 28.5937, Z -2.1667, A 0.000, B 0.000, C 0.000 }
gfCNCPoint2[732] = {X 269.2830, Y 28.5936, Z -2.1667, A 0.000, B 0.000, C 0.000 }
gfCNCPoint2[733] = {X 269.2829, Y 41.0279, Z -2.1667, A 0.000, B 0.000, C 0.000 }
gfCNCPoint2[734] = {X 269.3836, Y 41.1087, Z -2.1667, A 0.000, B 0.000, C 0.000 }
gfCNCPoint2[735] = {X 269.9800, Y 41.7409, Z -2.1667, A 0.000, B 0.000, C 0.000 }
gfCNCPoint2[736] = {X 270.4290, Y 42.4851, Z -2.1667, A 0.000, B 0.000, C 0.000 }
gfCNCPoint2[737] = {X 270.7102, Y 43.3075, Z -2.1667, A 0.000, B 0.000, C 0.000 }
gfCNCPoint2[738] = {X 270.8109, Y 44.1708, Z -2.1667, A 0.000, B 0.000, C 0.000 }
gfCNCPoint2[739] = {X 270.8110, Y 45.0000, Z -2.1667, A 0.000, B 0.000, C 0.000 }
gfCNCPoint2[740] = {X 270.7087, Y 45.9079, Z -2.1667, A 0.000, B 0.000, C 0.000 }
gfCNCPoint2[741] = {X 270.4070, Y 46.7702, Z -2.1667, A 0.000, B 0.000, C 0.000 }
gfCNCPoint2[742] = {X 269.9209, Y 47.5438, Z -2.1667, A 0.000, B 0.000, C 0.000 }
gfCNCPoint2[743] = {X 269.2749, Y 48.1899, Z -2.1667, A 0.000, B 0.000, C 0.000 }
gfCNCPoint2[744] = {X 268.5013, Y 48.6760, Z -2.1667, A 0.000, B 0.000, C 0.000 }
gfCNCPoint2[745] = {X 267.6389, Y 48.9777, Z -2.1667, A 0.000, B 0.000, C 0.000 }
gfCNCPoint2[746] = {X 266.7310, Y 49.0800, Z -2.1667, A 0.000, B 0.000, C 0.000 }
gfCNCPoint2[747] = {X 260.2876, Y 49.0800, Z -2.1667, A 0.000, B 0.000, C 0.000 }
gfCNCPoint2[748] = {X 259.3841, Y 48.9787, Z -2.1667, A 0.000, B 0.000, C 0.000 }
gfCNCPoint2[749] = {X 258.5255, Y 48.6799, Z -2.1667, A 0.000, B 0.000, C 0.000 }
gfCNCPoint2[750] = {X 257.7544, Y 48.1983, Z -2.1667, A 0.000, B 0.000, C 0.000 }
gfCNCPoint2[751] = {X 257.1090, Y 47.5580, Z -2.1667, A 0.000, B 0.000, C 0.000 }
gfCNCPoint2[752] = {X 256.6215, Y 46.7907, Z -2.1667, A 0.000, B 0.000, C 0.000 }
gfCNCPoint2[753] = {X 256.3160, Y 45.9344, Z -2.1667, A 0.000, B 0.000, C 0.000 }
gfCNCPoint2[754] = {X 256.2077, Y 45.0318, Z -2.1667, A 0.000, B 0.000, C 0.000 }
gfCNCPoint2[755] = {X 256.2080, Y 44.1527, Z -2.1667, A 0.000, B 0.000, C 0.000 }
gfCNCPoint2[756] = {X 256.3185, Y 43.2637, Z -2.1667, A 0.000, B 0.000, C 0.000 }
gfCNCPoint2[757] = {X 256.6204, Y 42.4203, Z -2.1667, A 0.000, B 0.000, C 0.000 }
gfCNCPoint2[758] = {X 257.0991, Y 41.6631, Z -2.1667, A 0.000, B 0.000, C 0.000 }
gfCNCPoint2[759] = {X 257.7315, Y 41.0287, Z -2.1667, A 0.000, B 0.000, C 0.000 }
gfCNCPoint2[760] = {X 257.7315, Y 34.2338, Z -2.1667, A 0.000, B 0.000, C 0.000 }
gfCNCPoint2[761] = {X 254.6202, Y 34.2338, Z -2.1667, A 0.000, B 0.000, C 0.000 }
gfCNCPoint2[762] = {X 250.2228, Y 42.8005, Z -2.1667, A 0.000, B 0.000, C 0.000 }
gfCNCPoint2[763] = {X 250.4073, Y 43.4766, Z -2.1667, A 0.000, B 0.000, C 0.000 }
gfCNCPoint2[764] = {X 250.4734, Y 44.1743, Z -2.1667, A 0.000, B 0.000, C 0.000 }
gfCNCPoint2[765] = {X 250.4736, Y 45.0000, Z -2.1667, A 0.000, B 0.000, C 0.000 }
gfCNCPoint2[766] = {X 250.3713, Y 45.9079, Z -2.1667, A 0.000, B 0.000, C 0.000 }
gfCNCPoint2[767] = {X 250.0695, Y 46.7702, Z -2.1667, A 0.000, B 0.000, C 0.000 }
gfCNCPoint2[768] = {X 249.5834, Y 47.5438, Z -2.1667, A 0.000, B 0.000, C 0.000 }
gfCNCPoint2[769] = {X 248.9374, Y 48.1899, Z -2.1667, A 0.000, B 0.000, C 0.000 }
gfCNCPoint2[770] = {X 248.1638, Y 48.6760, Z -2.1667, A 0.000, B 0.000, C 0.000 }
gfCNCPoint2[771] = {X 247.3014, Y 48.9777, Z -2.1667, A 0.000, B 0.000, C 0.000 }
gfCNCPoint2[772] = {X 246.3936, Y 49.0800, Z -2.1667, A 0.000, B 0.000, C 0.000 }
gfCNCPoint2[773] = {X 239.8075, Y 49.0800, Z -2.1667, A 0.000, B 0.000, C 0.000 }
gfCNCPoint2[774] = {X 238.8996, Y 48.9777, Z -2.1667, A 0.000, B 0.000, C 0.000 }
gfCNCPoint2[775] = {X 238.0373, Y 48.6760, Z -2.1667, A 0.000, B 0.000, C 0.000 }
gfCNCPoint2[776] = {X 237.2637, Y 48.1899, Z -2.1667, A 0.000, B 0.000, C 0.000 }
gfCNCPoint2[777] = {X 236.6176, Y 47.5438, Z -2.1667, A 0.000, B 0.000, C 0.000 }
gfCNCPoint2[778] = {X 236.1315, Y 46.7702, Z -2.1667, A 0.000, B 0.000, C 0.000 }
gfCNCPoint2[779] = {X 235.8298, Y 45.9079, Z -2.1667, A 0.000, B 0.000, C 0.000 }
gfCNCPoint2[780] = {X 235.7275, Y 45.0000, Z -2.1667, A 0.000, B 0.000, C 0.000 }
gfCNCPoint2[781] = {X 235.7279, Y 44.1527, Z -2.1667, A 0.000, B 0.000, C 0.000 }
gfCNCPoint2[782] = {X 235.8234, Y 43.3294, Z -2.1667, A 0.000, B 0.000, C 0.000 }
gfCNCPoint2[783] = {X 236.0833, Y 42.5424, Z -2.1667, A 0.000, B 0.000, C 0.000 }
gfCNCPoint2[784] = {X 236.4969, Y 41.8242, Z -2.1667, A 0.000, B 0.000, C 0.000 }
gfCNCPoint2[785] = {X 237.0471, Y 41.2044, Z -2.1667, A 0.000, B 0.000, C 0.000 }
gfCNCPoint2[786] = {X 237.7112, Y 40.7085, Z -2.1667, A 0.000, B 0.000, C 0.000 }
gfCNCPoint2[787] = {X 238.4618, Y 40.3571, Z -2.1667, A 0.000, B 0.000, C 0.000 }
gfCNCPoint2[788] = {X 242.5986, Y 32.2599, Z -2.1667, A 0.000, B 0.000, C 0.000 }
gfCNCPoint2[789] = {X 241.4076, Y 31.4914, Z -2.1667, A 0.000, B 0.000, C 0.000 }
gfCNCPoint2[790] = {X 240.3245, Y 30.5772, Z -2.1667, A 0.000, B 0.000, C 0.000 }
gfCNCPoint2[791] = {X 239.3671, Y 29.5321, Z -2.1667, A 0.000, B 0.000, C 0.000 }
gfCNCPoint2[792] = {X 238.5509, Y 28.3733, Z -2.1667, A 0.000, B 0.000, C 0.000 }
gfCNCPoint2[793] = {X 237.8894, Y 27.1198, Z -2.1667, A 0.000, B 0.000, C 0.000 }
gfCNCPoint2[794] = {X 237.3933, Y 25.7920, Z -2.1667, A 0.000, B 0.000, C 0.000 }
gfCNCPoint2[795] = {X 236.9796, Y 24.0072, Z -2.1667, A 0.000, B 0.000, C 0.000 }
gfCNCPoint2[796] = {X 236.7688, Y 22.1872, Z -2.1667, A 0.000, B 0.000, C 0.000 }
gfCNCPoint2[797] = {X 236.7637, Y 20.3551, Z -2.1667, A 0.000, B 0.000, C 0.000 }
gfCNCPoint2[798] = {X 236.9642, Y 18.5339, Z -2.1667, A 0.000, B 0.000, C 0.000 }
gfCNCPoint2[799] = {X 237.3680, Y 16.7468, Z -2.1667, A 0.000, B 0.000, C 0.000 }
gfCNCPoint2[800] = {X 237.9267, Y 15.2029, Z -2.1667, A 0.000, B 0.000, C 0.000 }
gfCNCPoint2[801] = {X 238.6977, Y 13.7534, Z -2.1667, A 0.000, B 0.000, C 0.000 }
gfCNCPoint2[802] = {X 239.6656, Y 12.4271, Z -2.1667, A 0.000, B 0.000, C 0.000 }
gfCNCPoint2[803] = {X 240.8110, Y 11.2507, Z -2.1667, A 0.000, B 0.000, C 0.000 }
gfCNCPoint2[804] = {X 242.1109, Y 10.2477, Z -2.1667, A 0.000, B 0.000, C 0.000 }
gfCNCPoint2[805] = {X 243.5393, Y 9.4382, Z -2.1667, A 0.000, B 0.000, C 0.000 }
gfCNCPoint2[806] = {X 245.0676, Y 8.8384, Z -2.1667, A 0.000, B 0.000, C 0.000 }
gfCNCPoint2[807] = {X 246.6653, Y 8.4602, Z -2.1667, A 0.000, B 0.000, C 0.000 }
gfCNCPoint2[808] = {X 248.7417, Y 8.1910, Z -2.1667, A 0.000, B 0.000, C 0.000 }
gfCNCPoint2[809] = {X 250.8340, Y 8.1116, Z -2.1667, A 0.000, B 0.000, C 0.000 }
gfCNCPoint2[810] = {X 266.7614, Y 8.1116, Z -2.1667, A 0.000, B 0.000, C 0.000 }
gfCNCPoint2[811] = {X 267.6634, Y 8.2200, Z -2.1667, A 0.000, B 0.000, C 0.000 }
gfCNCPoint2[812] = {X 268.5191, Y 8.5251, Z -2.1667, A 0.000, B 0.000, C 0.000 }
gfCNCPoint2[813] = {X 269.2861, Y 9.0120, Z -2.1667, A 0.000, B 0.000, C 0.000 }
gfCNCPoint2[814] = {X 269.9265, Y 9.6564, Z -2.1667, A 0.000, B 0.000, C 0.000 }
gfCNCPoint2[815] = {X 270.4085, Y 10.4265, Z -2.1667, A 0.000, B 0.000, C 0.000 }
gfCNCPoint2[816] = {X 270.7083, Y 11.2841, Z -2.1667, A 0.000, B 0.000, C 0.000 }
gfCNCPoint2[817] = {X 270.8110, Y 12.1867, Z -2.1667, A 0.000, B 0.000, C 0.000 }
gfCNCPoint2[818] = {X 270.8108, Y 13.0200, Z -2.1667, A 0.000, B 0.000, C 0.000 }
gfCNCPoint2[819] = {X 270.7022, Y 13.9140, Z -2.1667, A 0.000, B 0.000, C 0.000 }
gfCNCPoint2[820] = {X 270.4001, Y 14.7624, Z -2.1667, A 0.000, B 0.000, C 0.000 }
gfCNCPoint2[821] = {X 269.9193, Y 15.5239, Z -2.1667, A 0.000, B 0.000, C 0.000 }
gfCNCPoint2[822] = {X 269.2831, Y 16.1613, Z -2.1667, A 0.000, B 0.000, C 0.000 }
gfCNCPoint2[823] = {X 269.2830, Y 28.5936, Z -2.1667, A 0.000, B 0.000, C 0.000 }
gfCNCPoint2[824] = {X 273.2830, Y 28.5937, Z -2.1667, A 0.000, B 0.000, C 0.000 }
gfCNCPoint2[825] = {X 269.2030, Y 28.5936, Z -2.1667, A 0.000, B 0.000, C 0.000 }
gfCNCPoint2[826] = {X 269.2029, Y 41.0662, Z -2.1667, A 0.000, B 0.000, C 0.000 }
gfCNCPoint2[827] = {X 269.3419, Y 41.1783, Z -2.1667, A 0.000, B 0.000, C 0.000 }
gfCNCPoint2[828] = {X 269.9281, Y 41.8049, Z -2.1667, A 0.000, B 0.000, C 0.000 }
gfCNCPoint2[829] = {X 270.3672, Y 42.5420, Z -2.1667, A 0.000, B 0.000, C 0.000 }
gfCNCPoint2[830] = {X 270.6390, Y 43.3559, Z -2.1667, A 0.000, B 0.000, C 0.000 }
gfCNCPoint2[831] = {X 270.7310, Y 44.2089, Z -2.1667, A 0.000, B 0.000, C 0.000 }
gfCNCPoint2[832] = {X 270.7310, Y 45.0000, Z -2.1667, A 0.000, B 0.000, C 0.000 }
gfCNCPoint2[833] = {X 270.6307, Y 45.8901, Z -2.1667, A 0.000, B 0.000, C 0.000 }
gfCNCPoint2[834] = {X 270.3349, Y 46.7355, Z -2.1667, A 0.000, B 0.000, C 0.000 }
gfCNCPoint2[835] = {X 269.8584, Y 47.4940, Z -2.1667, A 0.000, B 0.000, C 0.000 }
gfCNCPoint2[836] = {X 269.2250, Y 48.1273, Z -2.1667, A 0.000, B 0.000, C 0.000 }
gfCNCPoint2[837] = {X 268.4666, Y 48.6039, Z -2.1667, A 0.000, B 0.000, C 0.000 }
gfCNCPoint2[838] = {X 267.6211, Y 48.8997, Z -2.1667, A 0.000, B 0.000, C 0.000 }
gfCNCPoint2[839] = {X 266.7310, Y 49.0000, Z -2.1667, A 0.000, B 0.000, C 0.000 }
gfCNCPoint2[840] = {X 260.2876, Y 49.0000, Z -2.1667, A 0.000, B 0.000, C 0.000 }
gfCNCPoint2[841] = {X 259.3975, Y 48.8997, Z -2.1667, A 0.000, B 0.000, C 0.000 }
gfCNCPoint2[842] = {X 258.5520, Y 48.6039, Z -2.1667, A 0.000, B 0.000, C 0.000 }
gfCNCPoint2[843] = {X 257.7936, Y 48.1273, Z -2.1667, A 0.000, B 0.000, C 0.000 }
gfCNCPoint2[844] = {X 257.1602, Y 47.4939, Z -2.1667, A 0.000, B 0.000, C 0.000 }
gfCNCPoint2[845] = {X 256.6837, Y 46.7355, Z -2.1667, A 0.000, B 0.000, C 0.000 }
gfCNCPoint2[846] = {X 256.3878, Y 45.8900, Z -2.1667, A 0.000, B 0.000, C 0.000 }
gfCNCPoint2[847] = {X 256.2876, Y 45.0000, Z -2.1667, A 0.000, B 0.000, C 0.000 }
gfCNCPoint2[848] = {X 256.2879, Y 44.1538, Z -2.1667, A 0.000, B 0.000, C 0.000 }
gfCNCPoint2[849] = {X 256.3986, Y 43.2730, Z -2.1667, A 0.000, B 0.000, C 0.000 }
gfCNCPoint2[850] = {X 256.7008, Y 42.4382, Z -2.1667, A 0.000, B 0.000, C 0.000 }
gfCNCPoint2[851] = {X 257.1796, Y 41.6907, Z -2.1667, A 0.000, B 0.000, C 0.000 }
gfCNCPoint2[852] = {X 257.8115, Y 41.0672, Z -2.1667, A 0.000, B 0.000, C 0.000 }
gfCNCPoint2[853] = {X 257.8115, Y 34.1538, Z -2.1667, A 0.000, B 0.000, C 0.000 }
gfCNCPoint2[854] = {X 254.8156, Y 34.1538, Z -2.1667, A 0.000, B 0.000, C 0.000 }
gfCNCPoint2[855] = {X 254.5726, Y 34.1514, Z -2.1667, A 0.000, B 0.000, C 0.000 }
gfCNCPoint2[856] = {X 250.1355, Y 42.7954, Z -2.1667, A 0.000, B 0.000, C 0.000 }
gfCNCPoint2[857] = {X 250.3285, Y 43.4905, Z -2.1667, A 0.000, B 0.000, C 0.000 }
gfCNCPoint2[858] = {X 250.3936, Y 44.2089, Z -2.1667, A 0.000, B 0.000, C 0.000 }
gfCNCPoint2[859] = {X 250.3936, Y 45.0000, Z -2.1667, A 0.000, B 0.000, C 0.000 }
gfCNCPoint2[860] = {X 250.2933, Y 45.8901, Z -2.1667, A 0.000, B 0.000, C 0.000 }
gfCNCPoint2[861] = {X 249.9974, Y 46.7355, Z -2.1667, A 0.000, B 0.000, C 0.000 }
gfCNCPoint2[862] = {X 249.5209, Y 47.4940, Z -2.1667, A 0.000, B 0.000, C 0.000 }
gfCNCPoint2[863] = {X 248.8875, Y 48.1273, Z -2.1667, A 0.000, B 0.000, C 0.000 }
gfCNCPoint2[864] = {X 248.1291, Y 48.6039, Z -2.1667, A 0.000, B 0.000, C 0.000 }
gfCNCPoint2[865] = {X 247.2836, Y 48.8997, Z -2.1667, A 0.000, B 0.000, C 0.000 }
gfCNCPoint2[866] = {X 246.3936, Y 49.0000, Z -2.1667, A 0.000, B 0.000, C 0.000 }
gfCNCPoint2[867] = {X 239.8075, Y 49.0000, Z -2.1667, A 0.000, B 0.000, C 0.000 }
gfCNCPoint2[868] = {X 238.9174, Y 48.8997, Z -2.1667, A 0.000, B 0.000, C 0.000 }
gfCNCPoint2[869] = {X 238.0720, Y 48.6039, Z -2.1667, A 0.000, B 0.000, C 0.000 }
gfCNCPoint2[870] = {X 237.3135, Y 48.1273, Z -2.1667, A 0.000, B 0.000, C 0.000 }
gfCNCPoint2[871] = {X 236.6802, Y 47.4940, Z -2.1667, A 0.000, B 0.000, C 0.000 }
gfCNCPoint2[872] = {X 236.2036, Y 46.7355, Z -2.1667, A 0.000, B 0.000, C 0.000 }
gfCNCPoint2[873] = {X 235.9078, Y 45.8901, Z -2.1667, A 0.000, B 0.000, C 0.000 }
gfCNCPoint2[874] = {X 235.8075, Y 45.0000, Z -2.1667, A 0.000, B 0.000, C 0.000 }
gfCNCPoint2[875] = {X 235.8079, Y 44.1538, Z -2.1667, A 0.000, B 0.000, C 0.000 }
gfCNCPoint2[876] = {X 235.9027, Y 43.3414, Z -2.1667, A 0.000, B 0.000, C 0.000 }
gfCNCPoint2[877] = {X 236.1607, Y 42.5654, Z -2.1667, A 0.000, B 0.000, C 0.000 }
gfCNCPoint2[878] = {X 236.5712, Y 41.8580, Z -2.1667, A 0.000, B 0.000, C 0.000 }
gfCNCPoint2[879] = {X 237.1169, Y 41.2489, Z -2.1667, A 0.000, B 0.000, C 0.000 }
gfCNCPoint2[880] = {X 237.7752, Y 40.7635, Z -2.1667, A 0.000, B 0.000, C 0.000 }
gfCNCPoint2[881] = {X 238.5184, Y 40.4222, Z -2.1667, A 0.000, B 0.000, C 0.000 }
gfCNCPoint2[882] = {X 242.7050, Y 32.2274, Z -2.1667, A 0.000, B 0.000, C 0.000 }
gfCNCPoint2[883] = {X 241.5070, Y 31.4652, Z -2.1667, A 0.000, B 0.000, C 0.000 }
gfCNCPoint2[884] = {X 240.4171, Y 30.5550, Z -2.1667, A 0.000, B 0.000, C 0.000 }
gfCNCPoint2[885] = {X 239.4536, Y 29.5119, Z -2.1667, A 0.000, B 0.000, C 0.000 }
gfCNCPoint2[886] = {X 238.6326, Y 28.3534, Z -2.1667, A 0.000, B 0.000, C 0.000 }
gfCNCPoint2[887] = {X 237.9676, Y 27.0987, Z -2.1667, A 0.000, B 0.000, C 0.000 }
gfCNCPoint2[888] = {X 237.4699, Y 25.7689, Z -2.1667, A 0.000, B 0.000, C 0.000 }
gfCNCPoint2[889] = {X 237.0583, Y 23.9929, Z -2.1667, A 0.000, B 0.000, C 0.000 }
gfCNCPoint2[890] = {X 236.8486, Y 22.1820, Z -2.1667, A 0.000, B 0.000, C 0.000 }
gfCNCPoint2[891] = {X 236.8436, Y 20.3590, Z -2.1667, A 0.000, B 0.000, C 0.000 }
gfCNCPoint2[892] = {X 237.0432, Y 18.5469, Z -2.1667, A 0.000, B 0.000, C 0.000 }
gfCNCPoint2[893] = {X 237.4449, Y 16.7687, Z -2.1667, A 0.000, B 0.000, C 0.000 }
gfCNCPoint2[894] = {X 237.9998, Y 15.2354, Z -2.1667, A 0.000, B 0.000, C 0.000 }
gfCNCPoint2[895] = {X 238.7656, Y 13.7958, Z -2.1667, A 0.000, B 0.000, C 0.000 }
gfCNCPoint2[896] = {X 239.7268, Y 12.4787, Z -2.1667, A 0.000, B 0.000, C 0.000 }
gfCNCPoint2[897] = {X 240.8643, Y 11.3103, Z -2.1667, A 0.000, B 0.000, C 0.000 }
gfCNCPoint2[898] = {X 242.1554, Y 10.3142, Z -2.1667, A 0.000, B 0.000, C 0.000 }
gfCNCPoint2[899] = {X 243.5740, Y 9.5103, Z -2.1667, A 0.000, B 0.000, C 0.000 }
gfCNCPoint2[900] = {X 245.0919, Y 8.9146, Z -2.1667, A 0.000, B 0.000, C 0.000 }
gfCNCPoint2[901] = {X 246.6787, Y 8.5391, Z -2.1667, A 0.000, B 0.000, C 0.000 }
gfCNCPoint2[902] = {X 248.7483, Y 8.2708, Z -2.1667, A 0.000, B 0.000, C 0.000 }
gfCNCPoint2[903] = {X 250.8336, Y 8.1916, Z -2.1667, A 0.000, B 0.000, C 0.000 }
gfCNCPoint2[904] = {X 266.7608, Y 8.1916, Z -2.1667, A 0.000, B 0.000, C 0.000 }
gfCNCPoint2[905] = {X 267.6451, Y 8.2978, Z -2.1667, A 0.000, B 0.000, C 0.000 }
gfCNCPoint2[906] = {X 268.4840, Y 8.5970, Z -2.1667, A 0.000, B 0.000, C 0.000 }
gfCNCPoint2[907] = {X 269.2360, Y 9.0743, Z -2.1667, A 0.000, B 0.000, C 0.000 }
gfCNCPoint2[908] = {X 269.8639, Y 9.7061, Z -2.1667, A 0.000, B 0.000, C 0.000 }
gfCNCPoint2[909] = {X 270.3364, Y 10.4611, Z -2.1667, A 0.000, B 0.000, C 0.000 }
gfCNCPoint2[910] = {X 270.6303, Y 11.3019, Z -2.1667, A 0.000, B 0.000, C 0.000 }
gfCNCPoint2[911] = {X 270.7310, Y 12.1869, Z -2.1667, A 0.000, B 0.000, C 0.000 }
gfCNCPoint2[912] = {X 270.7308, Y 13.0192, Z -2.1667, A 0.000, B 0.000, C 0.000 }
gfCNCPoint2[913] = {X 270.6221, Y 13.9050, Z -2.1667, A 0.000, B 0.000, C 0.000 }
gfCNCPoint2[914] = {X 270.3198, Y 14.7446, Z -2.1667, A 0.000, B 0.000, C 0.000 }
gfCNCPoint2[915] = {X 269.8388, Y 15.4963, Z -2.1667, A 0.000, B 0.000, C 0.000 }
gfCNCPoint2[916] = {X 269.2031, Y 16.1227, Z -2.1667, A 0.000, B 0.000, C 0.000 }
gfCNCPoint2[917] = {X 269.2030, Y 28.5936, Z -2.1667, A 0.000, B 0.000, C 0.000 }
gfCNCPoint2[918] = {X 273.2830, Y 28.5937, Z -2.1667, A 0.000, B 0.000, C 0.000 }
gfCNCPoint2[919] = {X 273.2830, Y 28.5937, Z 0.8333, A 0.000, B 0.000, C 0.000 }
gfCNCPoint2[920] = {X 273.2830, Y 28.5937, Z 11.0000, A 0.000, B 0.000, C 0.000 }
gfCNCPoint2[921] = {X 277.7460, Y 28.5931, Z 11.0000, A 0.000, B 0.000, C 0.000 }
gfCNCPoint2[922] = {X 277.7460, Y 28.5931, Z 0.8333, A 0.000, B 0.000, C 0.000 }
gfCNCPoint2[923] = {X 277.7460, Y 28.5931, Z -2.1667, A 0.000, B 0.000, C 0.000 }
gfCNCPoint2[924] = {X 281.8260, Y 28.5930, Z -2.1667, A 0.000, B 0.000, C 0.000 }
gfCNCPoint2[925] = {X 281.8258, Y 16.2747, Z -2.1667, A 0.000, B 0.000, C 0.000 }
gfCNCPoint2[926] = {X 281.1871, Y 15.6035, Z -2.1667, A 0.000, B 0.000, C 0.000 }
gfCNCPoint2[927] = {X 280.7061, Y 14.8116, Z -2.1667, A 0.000, B 0.000, C 0.000 }
gfCNCPoint2[928] = {X 280.4051, Y 13.9354, Z -2.1667, A 0.000, B 0.000, C 0.000 }
gfCNCPoint2[929] = {X 280.2978, Y 13.0151, Z -2.1667, A 0.000, B 0.000, C 0.000 }
gfCNCPoint2[930] = {X 280.2977, Y 12.1868, Z -2.1667, A 0.000, B 0.000, C 0.000 }
gfCNCPoint2[931] = {X 280.4060, Y 11.2255, Z -2.1667, A 0.000, B 0.000, C 0.000 }
gfCNCPoint2[932] = {X 280.7255, Y 10.3125, Z -2.1667, A 0.000, B 0.000, C 0.000 }
gfCNCPoint2[933] = {X 281.2402, Y 9.4933, Z -2.1667, A 0.000, B 0.000, C 0.000 }
gfCNCPoint2[934] = {X 281.9242, Y 8.8093, Z -2.1667, A 0.000, B 0.000, C 0.000 }
gfCNCPoint2[935] = {X 282.7433, Y 8.2946, Z -2.1667, A 0.000, B 0.000, C 0.000 }
gfCNCPoint2[936] = {X 283.6564, Y 7.9751, Z -2.1667, A 0.000, B 0.000, C 0.000 }
gfCNCPoint2[937] = {X 284.6177, Y 7.8668, Z -2.1667, A 0.000, B 0.000, C 0.000 }
gfCNCPoint2[938] = {X 291.0611, Y 7.8668, Z -2.1667, A 0.000, B 0.000, C 0.000 }
gfCNCPoint2[939] = {X 292.0224, Y 7.9751, Z -2.1667, A 0.000, B 0.000, C 0.000 }
gfCNCPoint2[940] = {X 292.9355, Y 8.2946, Z -2.1667, A 0.000, B 0.000, C 0.000 }
gfCNCPoint2[941] = {X 293.7546, Y 8.8093, Z -2.1667, A 0.000, B 0.000, C 0.000 }
gfCNCPoint2[942] = {X 294.4386, Y 9.4933, Z -2.1667, A 0.000, B 0.000, C 0.000 }
gfCNCPoint2[943] = {X 294.9533, Y 10.3124, Z -2.1667, A 0.000, B 0.000, C 0.000 }
gfCNCPoint2[944] = {X 295.2728, Y 11.2255, Z -2.1667, A 0.000, B 0.000, C 0.000 }
gfCNCPoint2[945] = {X 295.3811, Y 12.1868, Z -2.1667, A 0.000, B 0.000, C 0.000 }
gfCNCPoint2[946] = {X 295.3811, Y 12.9781, Z -2.1667, A 0.000, B 0.000, C 0.000 }
gfCNCPoint2[947] = {X 295.2797, Y 13.9083, Z -2.1667, A 0.000, B 0.000, C 0.000 }
gfCNCPoint2[948] = {X 294.9803, Y 14.7948, Z -2.1667, A 0.000, B 0.000, C 0.000 }
gfCNCPoint2[949] = {X 294.4971, Y 15.5961, Z -2.1667, A 0.000, B 0.000, C 0.000 }
gfCNCPoint2[950] = {X 293.8527, Y 16.2745, Z -2.1667, A 0.000, B 0.000, C 0.000 }
gfCNCPoint2[951] = {X 293.8540, Y 22.1965, Z -2.1667, A 0.000, B 0.000, C 0.000 }
gfCNCPoint2[952] = {X 302.7599, Y 22.1965, Z -2.1667, A 0.000, B 0.000, C 0.000 }
gfCNCPoint2[953] = {X 302.7646, Y 16.2783, Z -2.1667, A 0.000, B 0.000, C 0.000 }
gfCNCPoint2[954] = {X 302.1244, Y 15.6071, Z -2.1667, A 0.000, B 0.000, C 0.000 }
gfCNCPoint2[955] = {X 301.6422, Y 14.8148, Z -2.1667, A 0.000, B 0.000, C 0.000 }
gfCNCPoint2[956] = {X 301.3402, Y 13.9378, Z -2.1667, A 0.000, B 0.000, C 0.000 }
gfCNCPoint2[957] = {X 301.2324, Y 13.0165, Z -2.1667, A 0.000, B 0.000, C 0.000 }
gfCNCPoint2[958] = {X 301.2323, Y 12.1868, Z -2.1667, A 0.000, B 0.000, C 0.000 }
gfCNCPoint2[959] = {X 301.3406, Y 11.2255, Z -2.1667, A 0.000, B 0.000, C 0.000 }
gfCNCPoint2[960] = {X 301.6601, Y 10.3124, Z -2.1667, A 0.000, B 0.000, C 0.000 }
gfCNCPoint2[961] = {X 302.1747, Y 9.4933, Z -2.1667, A 0.000, B 0.000, C 0.000 }
gfCNCPoint2[962] = {X 302.8588, Y 8.8093, Z -2.1667, A 0.000, B 0.000, C 0.000 }
gfCNCPoint2[963] = {X 303.6779, Y 8.2946, Z -2.1667, A 0.000, B 0.000, C 0.000 }
gfCNCPoint2[964] = {X 304.5910, Y 7.9751, Z -2.1667, A 0.000, B 0.000, C 0.000 }
gfCNCPoint2[965] = {X 305.5523, Y 7.8668, Z -2.1667, A 0.000, B 0.000, C 0.000 }
gfCNCPoint2[966] = {X 311.9957, Y 7.8668, Z -2.1667, A 0.000, B 0.000, C 0.000 }
gfCNCPoint2[967] = {X 312.9570, Y 7.9751, Z -2.1667, A 0.000, B 0.000, C 0.000 }
gfCNCPoint2[968] = {X 313.8701, Y 8.2946, Z -2.1667, A 0.000, B 0.000, C 0.000 }
gfCNCPoint2[969] = {X 314.6892, Y 8.8093, Z -2.1667, A 0.000, B 0.000, C 0.000 }
gfCNCPoint2[970] = {X 315.3732, Y 9.4933, Z -2.1667, A 0.000, B 0.000, C 0.000 }
gfCNCPoint2[971] = {X 315.8879, Y 10.3124, Z -2.1667, A 0.000, B 0.000, C 0.000 }
gfCNCPoint2[972] = {X 316.2074, Y 11.2255, Z -2.1667, A 0.000, B 0.000, C 0.000 }
gfCNCPoint2[973] = {X 316.3157, Y 12.1868, Z -2.1667, A 0.000, B 0.000, C 0.000 }
gfCNCPoint2[974] = {X 316.3157, Y 12.9781, Z -2.1667, A 0.000, B 0.000, C 0.000 }
gfCNCPoint2[975] = {X 316.2144, Y 13.9084, Z -2.1667, A 0.000, B 0.000, C 0.000 }
gfCNCPoint2[976] = {X 315.9150, Y 14.7950, Z -2.1667, A 0.000, B 0.000, C 0.000 }
gfCNCPoint2[977] = {X 315.4319, Y 15.5963, Z -2.1667, A 0.000, B 0.000, C 0.000 }
gfCNCPoint2[978] = {X 314.7874, Y 16.2748, Z -2.1667, A 0.000, B 0.000, C 0.000 }
gfCNCPoint2[979] = {X 314.7872, Y 40.9118, Z -2.1667, A 0.000, B 0.000, C 0.000 }
gfCNCPoint2[980] = {X 315.4260, Y 41.5829, Z -2.1667, A 0.000, B 0.000, C 0.000 }
gfCNCPoint2[981] = {X 315.9071, Y 42.3748, Z -2.1667, A 0.000, B 0.000, C 0.000 }
gfCNCPoint2[982] = {X 316.2082, Y 43.2510, Z -2.1667, A 0.000, B 0.000, C 0.000 }
gfCNCPoint2[983] = {X 316.3156, Y 44.1713, Z -2.1667, A 0.000, B 0.000, C 0.000 }
gfCNCPoint2[984] = {X 316.3157, Y 45.0000, Z -2.1667, A 0.000, B 0.000, C 0.000 }
gfCNCPoint2[985] = {X 316.2074, Y 45.9613, Z -2.1667, A 0.000, B 0.000, C 0.000 }
gfCNCPoint2[986] = {X 315.8879, Y 46.8744, Z -2.1667, A 0.000, B 0.000, C 0.000 }
gfCNCPoint2[987] = {X 315.3732, Y 47.6935, Z -2.1667, A 0.000, B 0.000, C 0.000 }
gfCNCPoint2[988] = {X 314.6892, Y 48.3775, Z -2.1667, A 0.000, B 0.000, C 0.000 }
gfCNCPoint2[989] = {X 313.8701, Y 48.8922, Z -2.1667, A 0.000, B 0.000, C 0.000 }
gfCNCPoint2[990] = {X 312.9570, Y 49.2117, Z -2.1667, A 0.000, B 0.000, C 0.000 }
gfCNCPoint2[991] = {X 311.9957, Y 49.3200, Z -2.1667, A 0.000, B 0.000, C 0.000 }
gfCNCPoint2[992] = {X 305.5523, Y 49.3200, Z -2.1667, A 0.000, B 0.000, C 0.000 }
gfCNCPoint2[993] = {X 304.5958, Y 49.2128, Z -2.1667, A 0.000, B 0.000, C 0.000 }
gfCNCPoint2[994] = {X 303.6868, Y 48.8965, Z -2.1667, A 0.000, B 0.000, C 0.000 }
gfCNCPoint2[995] = {X 302.8704, Y 48.3868, Z -2.1667, A 0.000, B 0.000, C 0.000 }
gfCNCPoint2[996] = {X 302.1872, Y 47.7090, Z -2.1667, A 0.000, B 0.000, C 0.000 }
gfCNCPoint2[997] = {X 301.6709, Y 46.8967, Z -2.1667, A 0.000, B 0.000, C 0.000 }
gfCNCPoint2[998] = {X 301.3473, Y 45.9903, Z -2.1667, A 0.000, B 0.000, C 0.000 }
gfCNCPoint2[999] = {X 301.2324, Y 45.0348, Z -2.1667, A 0.000, B 0.000, C 0.000 }
gfCNCPoint2[1000] = {X 301.2324, Y 44.2011, Z -2.1667, A 0.000, B 0.000, C 0.000 }
gfCNCPoint2[1001] = {X 301.3504, Y 43.2650, Z -2.1667, A 0.000, B 0.000, C 0.000 }
gfCNCPoint2[1002] = {X 301.6539, Y 42.3717, Z -2.1667, A 0.000, B 0.000, C 0.000 }
gfCNCPoint2[1003] = {X 302.1305, Y 41.5575, Z -2.1667, A 0.000, B 0.000, C 0.000 }
gfCNCPoint2[1004] = {X 302.7607, Y 40.8554, Z -2.1667, A 0.000, B 0.000, C 0.000 }
gfCNCPoint2[1005] = {X 302.7607, Y 34.0343, Z -2.1667, A 0.000, B 0.000, C 0.000 }
gfCNCPoint2[1006] = {X 293.8537, Y 34.0343, Z -2.1667, A 0.000, B 0.000, C 0.000 }
gfCNCPoint2[1007] = {X 293.8528, Y 40.9028, Z -2.1667, A 0.000, B 0.000, C 0.000 }
gfCNCPoint2[1008] = {X 294.4918, Y 41.5867, Z -2.1667, A 0.000, B 0.000, C 0.000 }
gfCNCPoint2[1009] = {X 294.9725, Y 42.3898, Z -2.1667, A 0.000, B 0.000, C 0.000 }
gfCNCPoint2[1010] = {X 295.2735, Y 43.2762, Z -2.1667, A 0.000, B 0.000, C 0.000 }
gfCNCPoint2[1011] = {X 295.3811, Y 44.2060, Z -2.1667, A 0.000, B 0.000, C 0.000 }
gfCNCPoint2[1012] = {X 295.3811, Y 45.0000, Z -2.1667, A 0.000, B 0.000, C 0.000 }
gfCNCPoint2[1013] = {X 295.2728, Y 45.9613, Z -2.1667, A 0.000, B 0.000, C 0.000 }
gfCNCPoint2[1014] = {X 294.9533, Y 46.8744, Z -2.1667, A 0.000, B 0.000, C 0.000 }
gfCNCPoint2[1015] = {X 294.4386, Y 47.6935, Z -2.1667, A 0.000, B 0.000, C 0.000 }
gfCNCPoint2[1016] = {X 293.7546, Y 48.3775, Z -2.1667, A 0.000, B 0.000, C 0.000 }
gfCNCPoint2[1017] = {X 292.9355, Y 48.8922, Z -2.1667, A 0.000, B 0.000, C 0.000 }
gfCNCPoint2[1018] = {X 292.0224, Y 49.2117, Z -2.1667, A 0.000, B 0.000, C 0.000 }
gfCNCPoint2[1019] = {X 291.0611, Y 49.3200, Z -2.1667, A 0.000, B 0.000, C 0.000 }
gfCNCPoint2[1020] = {X 284.6177, Y 49.3200, Z -2.1667, A 0.000, B 0.000, C 0.000 }
gfCNCPoint2[1021] = {X 283.6613, Y 49.2128, Z -2.1667, A 0.000, B 0.000, C 0.000 }
gfCNCPoint2[1022] = {X 282.7524, Y 48.8965, Z -2.1667, A 0.000, B 0.000, C 0.000 }
gfCNCPoint2[1023] = {X 281.9360, Y 48.3869, Z -2.1667, A 0.000, B 0.000, C 0.000 }
gfCNCPoint2[1024] = {X 281.2527, Y 47.7092, Z -2.1667, A 0.000, B 0.000, C 0.000 }
gfCNCPoint2[1025] = {X 280.7365, Y 46.8970, Z -2.1667, A 0.000, B 0.000, C 0.000 }
gfCNCPoint2[1026] = {X 280.4128, Y 45.9907, Z -2.1667, A 0.000, B 0.000, C 0.000 }
gfCNCPoint2[1027] = {X 280.2978, Y 45.0352, Z -2.1667, A 0.000, B 0.000, C 0.000 }
gfCNCPoint2[1028] = {X 280.2977, Y 44.2070, Z -2.1667, A 0.000, B 0.000, C 0.000 }
gfCNCPoint2[1029] = {X 280.4031, Y 43.2782, Z -2.1667, A 0.000, B 0.000, C 0.000 }
gfCNCPoint2[1030] = {X 280.7035, Y 42.3929, Z -2.1667, A 0.000, B 0.000, C 0.000 }
gfCNCPoint2[1031] = {X 281.1852, Y 41.5918, Z -2.1667, A 0.000, B 0.000, C 0.000 }
gfCNCPoint2[1032] = {X 281.8262, Y 40.9113, Z -2.1667, A 0.000, B 0.000, C 0.000 }
gfCNCPoint2[1033] = {X 281.8260, Y 28.5930, Z -2.1667, A 0.000, B 0.000, C 0.000 }
gfCNCPoint2[1034] = {X 277.8260, Y 28.5931, Z -2.1667, A 0.000, B 0.000, C 0.000 }
gfCNCPoint2[1035] = {X 281.9060, Y 28.5930, Z -2.1667, A 0.000, B 0.000, C 0.000 }
gfCNCPoint2[1036] = {X 281.9058, Y 16.2374, Z -2.1667, A 0.000, B 0.000, C 0.000 }
gfCNCPoint2[1037] = {X 281.2675, Y 15.5769, Z -2.1667, A 0.000, B 0.000, C 0.000 }
gfCNCPoint2[1038] = {X 280.7864, Y 14.7944, Z -2.1667, A 0.000, B 0.000, C 0.000 }
gfCNCPoint2[1039] = {X 280.4852, Y 13.9267, Z -2.1667, A 0.000, B 0.000, C 0.000 }
gfCNCPoint2[1040] = {X 280.3778, Y 13.0144, Z -2.1667, A 0.000, B 0.000, C 0.000 }
gfCNCPoint2[1041] = {X 280.3777, Y 12.1868, Z -2.1667, A 0.000, B 0.000, C 0.000 }
gfCNCPoint2[1042] = {X 280.4840, Y 11.2433, Z -2.1667, A 0.000, B 0.000, C 0.000 }
gfCNCPoint2[1043] = {X 280.7976, Y 10.3472, Z -2.1667, A 0.000, B 0.000, C 0.000 }
gfCNCPoint2[1044] = {X 281.3027, Y 9.5432, Z -2.1667, A 0.000, B 0.000, C 0.000 }
gfCNCPoint2[1045] = {X 281.9741, Y 8.8719, Z -2.1667, A 0.000, B 0.000, C 0.000 }
gfCNCPoint2[1046] = {X 282.7780, Y 8.3667, Z -2.1667, A 0.000, B 0.000, C 0.000 }
gfCNCPoint2[1047] = {X 283.6742, Y 8.0531, Z -2.1667, A 0.000, B 0.000, C 0.000 }
gfCNCPoint2[1048] = {X 284.6177, Y 7.9468, Z -2.1667, A 0.000, B 0.000, C 0.000 }
gfCNCPoint2[1049] = {X 291.0611, Y 7.9468, Z -2.1667, A 0.000, B 0.000, C 0.000 }
gfCNCPoint2[1050] = {X 292.0046, Y 8.0531, Z -2.1667, A 0.000, B 0.000, C 0.000 }
gfCNCPoint2[1051] = {X 292.9008, Y 8.3667, Z -2.1667, A 0.000, B 0.000, C 0.000 }
gfCNCPoint2[1052] = {X 293.7047, Y 8.8718, Z -2.1667, A 0.000, B 0.000, C 0.000 }
gfCNCPoint2[1053] = {X 294.3761, Y 9.5432, Z -2.1667, A 0.000, B 0.000, C 0.000 }
gfCNCPoint2[1054] = {X 294.8812, Y 10.3471, Z -2.1667, A 0.000, B 0.000, C 0.000 }
gfCNCPoint2[1055] = {X 295.1948, Y 11.2433, Z -2.1667, A 0.000, B 0.000, C 0.000 }
gfCNCPoint2[1056] = {X 295.3011, Y 12.1868, Z -2.1667, A 0.000, B 0.000, C 0.000 }
gfCNCPoint2[1057] = {X 295.3011, Y 12.9781, Z -2.1667, A 0.000, B 0.000, C 0.000 }
gfCNCPoint2[1058] = {X 295.1996, Y 13.9001, Z -2.1667, A 0.000, B 0.000, C 0.000 }
gfCNCPoint2[1059] = {X 294.8999, Y 14.7779, Z -2.1667, A 0.000, B 0.000, C 0.000 }
gfCNCPoint2[1060] = {X 294.4166, Y 15.5696, Z -2.1667, A 0.000, B 0.000, C 0.000 }
gfCNCPoint2[1061] = {X 293.7727, Y 16.2372, Z -2.1667, A 0.000, B 0.000, C 0.000 }
gfCNCPoint2[1062] = {X 293.7740, Y 22.2765, Z -2.1667, A 0.000, B 0.000, C 0.000 }
gfCNCPoint2[1063] = {X 302.8398, Y 22.2765, Z -2.1667, A 0.000, B 0.000, C 0.000 }
gfCNCPoint2[1064] = {X 302.8447, Y 16.2409, Z -2.1667, A 0.000, B 0.000, C 0.000 }
gfCNCPoint2[1065] = {X 302.2049, Y 15.5804, Z -2.1667, A 0.000, B 0.000, C 0.000 }
gfCNCPoint2[1066] = {X 301.7225, Y 14.7975, Z -2.1667, A 0.000, B 0.000, C 0.000 }
gfCNCPoint2[1067] = {X 301.4203, Y 13.9290, Z -2.1667, A 0.000, B 0.000, C 0.000 }
gfCNCPoint2[1068] = {X 301.3124, Y 13.0158, Z -2.1667, A 0.000, B 0.000, C 0.000 }
gfCNCPoint2[1069] = {X 301.3123, Y 12.1868, Z -2.1667, A 0.000, B 0.000, C 0.000 }
gfCNCPoint2[1070] = {X 301.4186, Y 11.2433, Z -2.1667, A 0.000, B 0.000, C 0.000 }
gfCNCPoint2[1071] = {X 301.7321, Y 10.3471, Z -2.1667, A 0.000, B 0.000, C 0.000 }
gfCNCPoint2[1072] = {X 302.2373, Y 9.5432, Z -2.1667, A 0.000, B 0.000, C 0.000 }
gfCNCPoint2[1073] = {X 302.9087, Y 8.8718, Z -2.1667, A 0.000, B 0.000, C 0.000 }
gfCNCPoint2[1074] = {X 303.7126, Y 8.3667, Z -2.1667, A 0.000, B 0.000, C 0.000 }
gfCNCPoint2[1075] = {X 304.6088, Y 8.0531, Z -2.1667, A 0.000, B 0.000, C 0.000 }
gfCNCPoint2[1076] = {X 305.5523, Y 7.9468, Z -2.1667, A 0.000, B 0.000, C 0.000 }
gfCNCPoint2[1077] = {X 311.9957, Y 7.9468, Z -2.1667, A 0.000, B 0.000, C 0.000 }
gfCNCPoint2[1078] = {X 312.9392, Y 8.0531, Z -2.1667, A 0.000, B 0.000, C 0.000 }
gfCNCPoint2[1079] = {X 313.8354, Y 8.3667, Z -2.1667, A 0.000, B 0.000, C 0.000 }
gfCNCPoint2[1080] = {X 314.6393, Y 8.8718, Z -2.1667, A 0.000, B 0.000, C 0.000 }
gfCNCPoint2[1081] = {X 315.3107, Y 9.5432, Z -2.1667, A 0.000, B 0.000, C 0.000 }
gfCNCPoint2[1082] = {X 315.8158, Y 10.3471, Z -2.1667, A 0.000, B 0.000, C 0.000 }
gfCNCPoint2[1083] = {X 316.1294, Y 11.2433, Z -2.1667, A 0.000, B 0.000, C 0.000 }
gfCNCPoint2[1084] = {X 316.2357, Y 12.1868, Z -2.1667, A 0.000, B 0.000, C 0.000 }
gfCNCPoint2[1085] = {X 316.2357, Y 12.9781, Z -2.1667, A 0.000, B 0.000, C 0.000 }
gfCNCPoint2[1086] = {X 316.1342, Y 13.9002, Z -2.1667, A 0.000, B 0.000, C 0.000 }
gfCNCPoint2[1087] = {X 315.8347, Y 14.7781, Z -2.1667, A 0.000, B 0.000, C 0.000 }
gfCNCPoint2[1088] = {X 315.3514, Y 15.5698, Z -2.1667, A 0.000, B 0.000, C 0.000 }
gfCNCPoint2[1089] = {X 314.7074, Y 16.2375, Z -2.1667, A 0.000, B 0.000, C 0.000 }
gfCNCPoint2[1090] = {X 314.7072, Y 40.9504, Z -2.1667, A 0.000, B 0.000, C 0.000 }
gfCNCPoint2[1091] = {X 314.7355, Y 40.9729, Z -2.1667, A 0.000, B 0.000, C 0.000 }
gfCNCPoint2[1092] = {X 315.3625, Y 41.6315, Z -2.1667, A 0.000, B 0.000, C 0.000 }
gfCNCPoint2[1093] = {X 315.8346, Y 42.4087, Z -2.1667, A 0.000, B 0.000, C 0.000 }
gfCNCPoint2[1094] = {X 316.1302, Y 43.2687, Z -2.1667, A 0.000, B 0.000, C 0.000 }
gfCNCPoint2[1095] = {X 316.2356, Y 44.1720, Z -2.1667, A 0.000, B 0.000, C 0.000 }
gfCNCPoint2[1096] = {X 316.2357, Y 45.0000, Z -2.1667, A 0.000, B 0.000, C 0.000 }
gfCNCPoint2[1097] = {X 316.1294, Y 45.9435, Z -2.1667, A 0.000, B 0.000, C 0.000 }
gfCNCPoint2[1098] = {X 315.8158, Y 46.8397, Z -2.1667, A 0.000, B 0.000, C 0.000 }
gfCNCPoint2[1099] = {X 315.3107, Y 47.6436, Z -2.1667, A 0.000, B 0.000, C 0.000 }
gfCNCPoint2[1100] = {X 314.6393, Y 48.3150, Z -2.1667, A 0.000, B 0.000, C 0.000 }
gfCNCPoint2[1101] = {X 313.8354, Y 48.8201, Z -2.1667, A 0.000, B 0.000, C 0.000 }
gfCNCPoint2[1102] = {X 312.9392, Y 49.1337, Z -2.1667, A 0.000, B 0.000, C 0.000 }
gfCNCPoint2[1103] = {X 311.9957, Y 49.2400, Z -2.1667, A 0.000, B 0.000, C 0.000 }
gfCNCPoint2[1104] = {X 305.5523, Y 49.2400, Z -2.1667, A 0.000, B 0.000, C 0.000 }
gfCNCPoint2[1105] = {X 304.6135, Y 49.1348, Z -2.1667, A 0.000, B 0.000, C 0.000 }
gfCNCPoint2[1106] = {X 303.7214, Y 48.8243, Z -2.1667, A 0.000, B 0.000, C 0.000 }
gfCNCPoint2[1107] = {X 302.9201, Y 48.3241, Z -2.1667, A 0.000, B 0.000, C 0.000 }
gfCNCPoint2[1108] = {X 302.2495, Y 47.6588, Z -2.1667, A 0.000, B 0.000, C 0.000 }
gfCNCPoint2[1109] = {X 301.7428, Y 46.8616, Z -2.1667, A 0.000, B 0.000, C 0.000 }
gfCNCPoint2[1110] = {X 301.4252, Y 45.9720, Z -2.1667, A 0.000, B 0.000, C 0.000 }
gfCNCPoint2[1111] = {X 301.3124, Y 45.0341, Z -2.1667, A 0.000, B 0.000, C 0.000 }
gfCNCPoint2[1112] = {X 301.3123, Y 44.2030, Z -2.1667, A 0.000, B 0.000, C 0.000 }
gfCNCPoint2[1113] = {X 301.4304, Y 43.2744, Z -2.1667, A 0.000, B 0.000, C 0.000 }
gfCNCPoint2[1114] = {X 301.7340, Y 42.3889, Z -2.1667, A 0.000, B 0.000, C 0.000 }
gfCNCPoint2[1115] = {X 302.2108, Y 41.5833, Z -2.1667, A 0.000, B 0.000, C 0.000 }
gfCNCPoint2[1116] = {X 302.8407, Y 40.8909, Z -2.1667, A 0.000, B 0.000, C 0.000 }
gfCNCPoint2[1117] = {X 302.8407, Y 33.9543, Z -2.1667, A 0.000, B 0.000, C 0.000 }
gfCNCPoint2[1118] = {X 293.7738, Y 33.9543, Z -2.1667, A 0.000, B 0.000, C 0.000 }
gfCNCPoint2[1119] = {X 293.7728, Y 40.9395, Z -2.1667, A 0.000, B 0.000, C 0.000 }
gfCNCPoint2[1120] = {X 294.4114, Y 41.6131, Z -2.1667, A 0.000, B 0.000, C 0.000 }
gfCNCPoint2[1121] = {X 294.8922, Y 42.4069, Z -2.1667, A 0.000, B 0.000, C 0.000 }
gfCNCPoint2[1122] = {X 295.1934, Y 43.2848, Z -2.1667, A 0.000, B 0.000, C 0.000 }
gfCNCPoint2[1123] = {X 295.3011, Y 44.2067, Z -2.1667, A 0.000, B 0.000, C 0.000 }
gfCNCPoint2[1124] = {X 295.3011, Y 45.0000, Z -2.1667, A 0.000, B 0.000, C 0.000 }
gfCNCPoint2[1125] = {X 295.1948, Y 45.9435, Z -2.1667, A 0.000, B 0.000, C 0.000 }
gfCNCPoint2[1126] = {X 294.8812, Y 46.8397, Z -2.1667, A 0.000, B 0.000, C 0.000 }
gfCNCPoint2[1127] = {X 294.3761, Y 47.6436, Z -2.1667, A 0.000, B 0.000, C 0.000 }
gfCNCPoint2[1128] = {X 293.7047, Y 48.3150, Z -2.1667, A 0.000, B 0.000, C 0.000 }
gfCNCPoint2[1129] = {X 292.9008, Y 48.8201, Z -2.1667, A 0.000, B 0.000, C 0.000 }
gfCNCPoint2[1130] = {X 292.0046, Y 49.1337, Z -2.1667, A 0.000, B 0.000, C 0.000 }
gfCNCPoint2[1131] = {X 291.0611, Y 49.2400, Z -2.1667, A 0.000, B 0.000, C 0.000 }
gfCNCPoint2[1132] = {X 284.6177, Y 49.2400, Z -2.1667, A 0.000, B 0.000, C 0.000 }
gfCNCPoint2[1133] = {X 283.6790, Y 49.1348, Z -2.1667, A 0.000, B 0.000, C 0.000 }
gfCNCPoint2[1134] = {X 282.7869, Y 48.8244, Z -2.1667, A 0.000, B 0.000, C 0.000 }
gfCNCPoint2[1135] = {X 281.9857, Y 48.3242, Z -2.1667, A 0.000, B 0.000, C 0.000 }
gfCNCPoint2[1136] = {X 281.3150, Y 47.6590, Z -2.1667, A 0.000, B 0.000, C 0.000 }
gfCNCPoint2[1137] = {X 280.8083, Y 46.8619, Z -2.1667, A 0.000, B 0.000, C 0.000 }
gfCNCPoint2[1138] = {X 280.4907, Y 45.9723, Z -2.1667, A 0.000, B 0.000, C 0.000 }
gfCNCPoint2[1139] = {X 280.3778, Y 45.0345, Z -2.1667, A 0.000, B 0.000, C 0.000 }
gfCNCPoint2[1140] = {X 280.3777, Y 44.2075, Z -2.1667, A 0.000, B 0.000, C 0.000 }
gfCNCPoint2[1141] = {X 280.4832, Y 43.2867, Z -2.1667, A 0.000, B 0.000, C 0.000 }
gfCNCPoint2[1142] = {X 280.7838, Y 42.4100, Z -2.1667, A 0.000, B 0.000, C 0.000 }
gfCNCPoint2[1143] = {X 281.2657, Y 41.6182, Z -2.1667, A 0.000, B 0.000, C 0.000 }
gfCNCPoint2[1144] = {X 281.9062, Y 40.9484, Z -2.1667, A 0.000, B 0.000, C 0.000 }
gfCNCPoint2[1145] = {X 281.9060, Y 28.5930, Z -2.1667, A 0.000, B 0.000, C 0.000 }
gfCNCPoint2[1146] = {X 277.9060, Y 28.5931, Z -2.1667, A 0.000, B 0.000, C 0.000 }
gfCNCPoint2[1147] = {X 281.9860, Y 28.5930, Z -2.1667, A 0.000, B 0.000, C 0.000 }
gfCNCPoint2[1148] = {X 281.9858, Y 16.1997, Z -2.1667, A 0.000, B 0.000, C 0.000 }
gfCNCPoint2[1149] = {X 281.3480, Y 15.5499, Z -2.1667, A 0.000, B 0.000, C 0.000 }
gfCNCPoint2[1150] = {X 280.8668, Y 14.7770, Z -2.1667, A 0.000, B 0.000, C 0.000 }
gfCNCPoint2[1151] = {X 280.5652, Y 13.9179, Z -2.1667, A 0.000, B 0.000, C 0.000 }
gfCNCPoint2[1152] = {X 280.4578, Y 13.0137, Z -2.1667, A 0.000, B 0.000, C 0.000 }
gfCNCPoint2[1153] = {X 280.4577, Y 12.1868, Z -2.1667, A 0.000, B 0.000, C 0.000 }
gfCNCPoint2[1154] = {X 280.5620, Y 11.2611, Z -2.1667, A 0.000, B 0.000, C 0.000 }
gfCNCPoint2[1155] = {X 280.8696, Y 10.3819, Z -2.1667, A 0.000, B 0.000, C 0.000 }
gfCNCPoint2[1156] = {X 281.3652, Y 9.5931, Z -2.1667, A 0.000, B 0.000, C 0.000 }
gfCNCPoint2[1157] = {X 282.0240, Y 8.9344, Z -2.1667, A 0.000, B 0.000, C 0.000 }
gfCNCPoint2[1158] = {X 282.8127, Y 8.4388, Z -2.1667, A 0.000, B 0.000, C 0.000 }
gfCNCPoint2[1159] = {X 283.6920, Y 8.1311, Z -2.1667, A 0.000, B 0.000, C 0.000 }
gfCNCPoint2[1160] = {X 284.6177, Y 8.0268, Z -2.1667, A 0.000, B 0.000, C 0.000 }
gfCNCPoint2[1161] = {X 291.0611, Y 8.0268, Z -2.1667, A 0.000, B 0.000, C 0.000 }
gfCNCPoint2[1162] = {X 291.9868, Y 8.1311, Z -2.1667, A 0.000, B 0.000, C 0.000 }
gfCNCPoint2[1163] = {X 292.8661, Y 8.4388, Z -2.1667, A 0.000, B 0.000, C 0.000 }
gfCNCPoint2[1164] = {X 293.6549, Y 8.9344, Z -2.1667, A 0.000, B 0.000, C 0.000 }
gfCNCPoint2[1165] = {X 294.3136, Y 9.5931, Z -2.1667, A 0.000, B 0.000, C 0.000 }
gfCNCPoint2[1166] = {X 294.8092, Y 10.3819, Z -2.1667, A 0.000, B 0.000, C 0.000 }
gfCNCPoint2[1167] = {X 295.1168, Y 11.2611, Z -2.1667, A 0.000, B 0.000, C 0.000 }
gfCNCPoint2[1168] = {X 295.2211, Y 12.1868, Z -2.1667, A 0.000, B 0.000, C 0.000 }
gfCNCPoint2[1169] = {X 295.2211, Y 12.9781, Z -2.1667, A 0.000, B 0.000, C 0.000 }
gfCNCPoint2[1170] = {X 295.1254, Y 13.8654, Z -2.1667, A 0.000, B 0.000, C 0.000 }
gfCNCPoint2[1171] = {X 294.8426, Y 14.7118, Z -2.1667, A 0.000, B 0.000, C 0.000 }
gfCNCPoint2[1172] = {X 294.3858, Y 15.4784, Z -2.1667, A 0.000, B 0.000, C 0.000 }
gfCNCPoint2[1173] = {X 293.7761, Y 16.1300, Z -2.1667, A 0.000, B 0.000, C 0.000 }
gfCNCPoint2[1174] = {X 293.6927, Y 16.1999, Z -2.1667, A 0.000, B 0.000, C 0.000 }
gfCNCPoint2[1175] = {X 293.6940, Y 22.3568, Z -2.1667, A 0.000, B 0.000, C 0.000 }
gfCNCPoint2[1176] = {X 302.9197, Y 22.3565, Z -2.1667, A 0.000, B 0.000, C 0.000 }
gfCNCPoint2[1177] = {X 302.9247, Y 16.2032, Z -2.1667, A 0.000, B 0.000, C 0.000 }
gfCNCPoint2[1178] = {X 302.2853, Y 15.5535, Z -2.1667, A 0.000, B 0.000, C 0.000 }
gfCNCPoint2[1179] = {X 301.8028, Y 14.7801, Z -2.1667, A 0.000, B 0.000, C 0.000 }
gfCNCPoint2[1180] = {X 301.5004, Y 13.9202, Z -2.1667, A 0.000, B 0.000, C 0.000 }
gfCNCPoint2[1181] = {X 301.3924, Y 13.0151, Z -2.1667, A 0.000, B 0.000, C 0.000 }
gfCNCPoint2[1182] = {X 301.3923, Y 12.1868, Z -2.1667, A 0.000, B 0.000, C 0.000 }
gfCNCPoint2[1183] = {X 301.4966, Y 11.2611, Z -2.1667, A 0.000, B 0.000, C 0.000 }
gfCNCPoint2[1184] = {X 301.8042, Y 10.3819, Z -2.1667, A 0.000, B 0.000, C 0.000 }
gfCNCPoint2[1185] = {X 302.2998, Y 9.5931, Z -2.1667, A 0.000, B 0.000, C 0.000 }
gfCNCPoint2[1186] = {X 302.9585, Y 8.9344, Z -2.1667, A 0.000, B 0.000, C 0.000 }
gfCNCPoint2[1187] = {X 303.7473, Y 8.4388, Z -2.1667, A 0.000, B 0.000, C 0.000 }
gfCNCPoint2[1188] = {X 304.6266, Y 8.1311, Z -2.1667, A 0.000, B 0.000, C 0.000 }
gfCNCPoint2[1189] = {X 305.5523, Y 8.0268, Z -2.1667, A 0.000, B 0.000, C 0.000 }
gfCNCPoint2[1190] = {X 311.9957, Y 8.0268, Z -2.1667, A 0.000, B 0.000, C 0.000 }
gfCNCPoint2[1191] = {X 312.9214, Y 8.1311, Z -2.1667, A 0.000, B 0.000, C 0.000 }
gfCNCPoint2[1192] = {X 313.8007, Y 8.4388, Z -2.1667, A 0.000, B 0.000, C 0.000 }
gfCNCPoint2[1193] = {X 314.5894, Y 8.9344, Z -2.1667, A 0.000, B 0.000, C 0.000 }
gfCNCPoint2[1194] = {X 315.2481, Y 9.5931, Z -2.1667, A 0.000, B 0.000, C 0.000 }
gfCNCPoint2[1195] = {X 315.7438, Y 10.3819, Z -2.1667, A 0.000, B 0.000, C 0.000 }
gfCNCPoint2[1196] = {X 316.0514, Y 11.2611, Z -2.1667, A 0.000, B 0.000, C 0.000 }
gfCNCPoint2[1197] = {X 316.1557, Y 12.1868, Z -2.1667, A 0.000, B 0.000, C 0.000 }
gfCNCPoint2[1198] = {X 316.1557, Y 12.9781, Z -2.1667, A 0.000, B 0.000, C 0.000 }
gfCNCPoint2[1199] = {X 316.0541, Y 13.8917, Z -2.1667, A 0.000, B 0.000, C 0.000 }
gfCNCPoint2[1200] = {X 315.7544, Y 14.7606, Z -2.1667, A 0.000, B 0.000, C 0.000 }
gfCNCPoint2[1201] = {X 315.2712, Y 15.5425, Z -2.1667, A 0.000, B 0.000, C 0.000 }
gfCNCPoint2[1202] = {X 314.6281, Y 16.1993, Z -2.1667, A 0.000, B 0.000, C 0.000 }
gfCNCPoint2[1203] = {X 314.6272, Y 40.9893, Z -2.1667, A 0.000, B 0.000, C 0.000 }
gfCNCPoint2[1204] = {X 314.6831, Y 41.0334, Z -2.1667, A 0.000, B 0.000, C 0.000 }
gfCNCPoint2[1205] = {X 315.2986, Y 41.6796, Z -2.1667, A 0.000, B 0.000, C 0.000 }
gfCNCPoint2[1206] = {X 315.7620, Y 42.4423, Z -2.1667, A 0.000, B 0.000, C 0.000 }
gfCNCPoint2[1207] = {X 316.0521, Y 43.2862, Z -2.1667, A 0.000, B 0.000, C 0.000 }
gfCNCPoint2[1208] = {X 316.1556, Y 44.1727, Z -2.1667, A 0.000, B 0.000, C 0.000 }
gfCNCPoint2[1209] = {X 316.1557, Y 45.0000, Z -2.1667, A 0.000, B 0.000, C 0.000 }
gfCNCPoint2[1210] = {X 316.0514, Y 45.9257, Z -2.1667, A 0.000, B 0.000, C 0.000 }
gfCNCPoint2[1211] = {X 315.7438, Y 46.8050, Z -2.1667, A 0.000, B 0.000, C 0.000 }
gfCNCPoint2[1212] = {X 315.2481, Y 47.5937, Z -2.1667, A 0.000, B 0.000, C 0.000 }
gfCNCPoint2[1213] = {X 314.5894, Y 48.2524, Z -2.1667, A 0.000, B 0.000, C 0.000 }
gfCNCPoint2[1214] = {X 313.8007, Y 48.7480, Z -2.1667, A 0.000, B 0.000, C 0.000 }
gfCNCPoint2[1215] = {X 312.9214, Y 49.0557, Z -2.1667, A 0.000, B 0.000, C 0.000 }
gfCNCPoint2[1216] = {X 311.9957, Y 49.1600, Z -2.1667, A 0.000, B 0.000, C 0.000 }
gfCNCPoint2[1217] = {X 305.5523, Y 49.1600, Z -2.1667, A 0.000, B 0.000, C 0.000 }
gfCNCPoint2[1218] = {X 304.6312, Y 49.0568, Z -2.1667, A 0.000, B 0.000, C 0.000 }
gfCNCPoint2[1219] = {X 303.7559, Y 48.7522, Z -2.1667, A 0.000, B 0.000, C 0.000 }
